   LIN {X 10.637, Y -21.360, Z 102.000}
   LaserEnd_Ext()
   LIN {X 11.146, Y -20.360, Z 102.000}
   LaserStart_Ext()
   LIN {X 9.029, Y -20.360, Z 102.000}
   LaserEnd_Ext()
   LIN {X -1.745, Y -20.360, Z 102.000}
   LaserStart_Ext()
   LIN {X -3.794, Y -20.360, Z 102.000}
   LaserEnd_Ext()
   LIN {X -4.048, Y -19.360, Z 102.000}
   LaserStart_Ext()
   LIN {X -2.060, Y -19.360, Z 102.000}
   LaserEnd_Ext()
   LIN {X 9.299, Y -19.360, Z 102.000}
   LaserStart_Ext()
   LIN {X 11.371, Y -19.360, Z 102.000}
   LaserEnd_Ext()
   LIN {X 11.596, Y -18.360, Z 102.000}
   LaserStart_Ext()
   LIN {X 9.570, Y -18.360, Z 102.000}
   LaserEnd_Ext()
   LIN {X -2.335, Y -18.360, Z 102.000}
   LaserStart_Ext()
   LIN {X -4.308, Y -18.360, Z 102.000}
   LaserEnd_Ext()
   LIN {X -4.240, Y -17.360, Z 102.000}
   LaserStart_Ext()
   LIN {X -2.147, Y -17.360, Z 102.000}
   LaserEnd_Ext()
   LIN {X 9.558, Y -17.360, Z 102.000}
   LaserStart_Ext()
   LIN {X 11.679, Y -17.360, Z 102.000}
   LaserEnd_Ext()
   LIN {X 11.721, Y -16.360, Z 102.000}
   LaserStart_Ext()
   LIN {X 9.366, Y -16.360, Z 102.000}
   LaserEnd_Ext()
   LIN {X -1.926, Y -16.360, Z 102.000}
   LaserStart_Ext()
   LIN {X -4.108, Y -16.360, Z 102.000}
   LaserEnd_Ext()
   LIN {X -3.973, Y -15.360, Z 102.000}
   LaserStart_Ext()
   LIN {X -1.705, Y -15.360, Z 102.000}
   LaserEnd_Ext()
   LIN {X 9.145, Y -15.360, Z 102.000}
   LaserStart_Ext()
   LIN {X 11.764, Y -15.360, Z 102.000}
   LaserEnd_Ext()
   LIN {X 11.791, Y -14.360, Z 102.000}
   LaserStart_Ext()
   LIN {X 8.388, Y -14.360, Z 102.000}
   LaserEnd_Ext()
   LIN {X -1.169, Y -14.360, Z 102.000}
   LaserStart_Ext()
   LIN {X -3.678, Y -14.360, Z 102.000}
   LaserEnd_Ext()
   LIN {X -3.386, Y -13.360, Z 102.000}
   LaserStart_Ext()
   LIN {X -0.277, Y -13.360, Z 102.000}
   LaserEnd_Ext()
   LIN {X 7.590, Y -13.360, Z 102.000}
   LaserStart_Ext()
   LIN {X 11.806, Y -13.360, Z 102.000}
   LaserEnd_Ext()
   LIN {X 11.817, Y -12.360, Z 102.000}
   LaserStart_Ext()
   LIN {X 5.937, Y -12.360, Z 102.000}
   LaserEnd_Ext()
   LIN {X 1.421, Y -12.360, Z 102.000}
   LaserStart_Ext()
   LIN {X -3.094, Y -12.360, Z 102.000}
   LaserEnd_Ext()
   LIN {X -2.845, Y -11.360, Z 102.000}
   LaserStart_Ext()
   LIN {X 11.809, Y -11.360, Z 102.000}
   LaserEnd_Ext()
   LIN {X 11.793, Y -10.360, Z 102.000}
   LaserStart_Ext()
   LIN {X -2.605, Y -10.360, Z 102.000}
   LaserEnd_Ext()
   LIN {X -2.364, Y -9.360, Z 102.000}
   LaserStart_Ext()
   LIN {X 11.776, Y -9.360, Z 102.000}
   LaserEnd_Ext()
   LIN {X 11.758, Y -8.360, Z 102.000}
   LaserStart_Ext()
   LIN {X -2.129, Y -8.360, Z 102.000}
   LaserEnd_Ext()
   LIN {X -1.924, Y -7.360, Z 102.000}
   LaserStart_Ext()
   LIN {X 11.706, Y -7.360, Z 102.000}
   LaserEnd_Ext()
   LIN {X 11.652, Y -6.360, Z 102.000}
   LaserStart_Ext()
   LIN {X -1.769, Y -6.360, Z 102.000}
   LaserEnd_Ext()
   LIN {X -1.619, Y -5.360, Z 102.000}
   LaserStart_Ext()
   LIN {X 11.597, Y -5.360, Z 102.000}
   LaserEnd_Ext()
   LIN {X 11.543, Y -4.360, Z 102.000}
   LaserStart_Ext()
   LIN {X -1.468, Y -4.360, Z 102.000}
   LaserEnd_Ext()
   LIN {X -1.317, Y -3.360, Z 102.000}
   LaserStart_Ext()
   LIN {X 11.470, Y -3.360, Z 102.000}
   LaserEnd_Ext()
   LIN {X 11.369, Y -2.360, Z 102.000}
   LaserStart_Ext()
   LIN {X -1.166, Y -2.360, Z 102.000}
   LaserEnd_Ext()
   LIN {X -1.015, Y -1.360, Z 102.000}
   LaserStart_Ext()
   LIN {X 11.269, Y -1.360, Z 102.000}
   LaserEnd_Ext()
   LIN {X 11.168, Y -0.360, Z 102.000}
   LaserStart_Ext()
   LIN {X -0.870, Y -0.360, Z 102.000}
   LaserEnd_Ext()
   LIN {X -0.832, Y 0.640, Z 102.000}
   LaserStart_Ext()
   LIN {X 11.068, Y 0.640, Z 102.000}
   LaserEnd_Ext()
   LIN {X 10.962, Y 1.640, Z 102.000}
   LaserStart_Ext()
   LIN {X -0.795, Y 1.640, Z 102.000}
   LaserEnd_Ext()
   LIN {X -0.758, Y 2.640, Z 102.000}
   LaserStart_Ext()
   LIN {X 10.799, Y 2.640, Z 102.000}
   LaserEnd_Ext()
   LIN {X 10.635, Y 3.640, Z 102.000}
   LaserStart_Ext()
   LIN {X -0.721, Y 3.640, Z 102.000}
   LaserEnd_Ext()
   LIN {X -0.684, Y 4.640, Z 102.000}
   LaserStart_Ext()
   LIN {X 10.471, Y 4.640, Z 102.000}
   LaserEnd_Ext()
   LIN {X 10.308, Y 5.640, Z 102.000}
   LaserStart_Ext()
   LIN {X -0.647, Y 5.640, Z 102.000}
   LaserEnd_Ext()
   LIN {X -0.610, Y 6.640, Z 102.000}
   LaserStart_Ext()
   LIN {X 10.144, Y 6.640, Z 102.000}
   LaserEnd_Ext()
   LIN {X 9.981, Y 7.640, Z 102.000}
   LaserStart_Ext()
   LIN {X -0.570, Y 7.640, Z 102.000}
   LaserEnd_Ext()
   LIN {X -0.514, Y 8.640, Z 102.000}
   LaserStart_Ext()
   LIN {X 9.817, Y 8.640, Z 102.000}
   LaserEnd_Ext()
   LIN {X 9.654, Y 9.640, Z 102.000}
   LaserStart_Ext()
   LIN {X -0.579, Y 9.640, Z 102.000}
   LaserEnd_Ext()
   LIN {X -0.671, Y 10.640, Z 102.000}
   LaserStart_Ext()
   LIN {X 9.429, Y 10.640, Z 102.000}
   LaserEnd_Ext()
   LIN {X 9.178, Y 11.640, Z 102.000}
   LaserStart_Ext()
   LIN {X -0.763, Y 11.640, Z 102.000}
   LaserEnd_Ext()
   LIN {X -0.856, Y 12.640, Z 102.000}
   LaserStart_Ext()
   LIN {X 8.927, Y 12.640, Z 102.000}
   LaserEnd_Ext()
   LIN {X 8.677, Y 13.640, Z 102.000}
   LaserStart_Ext()
   LIN {X -0.948, Y 13.640, Z 102.000}
   LaserEnd_Ext()
   LIN {X -1.040, Y 14.640, Z 102.000}
   LaserStart_Ext()
   LIN {X 8.426, Y 14.640, Z 102.000}
   LaserEnd_Ext()
   LIN {X 8.175, Y 15.640, Z 102.000}
   LaserStart_Ext()
   LIN {X -1.132, Y 15.640, Z 102.000}
   LaserEnd_Ext()
   LIN {X -1.224, Y 16.640, Z 102.000}
   LaserStart_Ext()
   LIN {X 7.925, Y 16.640, Z 102.000}
   LaserEnd_Ext()
   LIN {X 7.674, Y 17.640, Z 102.000}
   LaserStart_Ext()
   LIN {X -1.316, Y 17.640, Z 102.000}
   LaserEnd_Ext()
   LIN {X -1.415, Y 18.640, Z 102.000}
   LaserStart_Ext()
   LIN {X 7.428, Y 18.640, Z 102.000}
   LaserEnd_Ext()
   LIN {X 7.127, Y 19.640, Z 102.000}
   LaserStart_Ext()
   LIN {X -1.612, Y 19.640, Z 102.000}
   LaserEnd_Ext()
   LIN {X -1.838, Y 20.640, Z 102.000}
   LaserStart_Ext()
   LIN {X 6.799, Y 20.640, Z 102.000}
   LaserEnd_Ext()
   LIN {X 6.471, Y 21.640, Z 102.000}
   LaserStart_Ext()
   LIN {X -2.067, Y 21.640, Z 102.000}
   LaserEnd_Ext()
   LIN {X -2.296, Y 22.640, Z 102.000}
   LaserStart_Ext()
   LIN {X 6.144, Y 22.640, Z 102.000}
   LaserEnd_Ext()
   LIN {X 5.816, Y 23.640, Z 102.000}
   LaserStart_Ext()
   LIN {X -2.517, Y 23.640, Z 102.000}
   LaserEnd_Ext()
   LIN {X -2.736, Y 24.640, Z 102.000}
   LaserStart_Ext()
   LIN {X 5.488, Y 24.640, Z 102.000}
   LaserEnd_Ext()
   LIN {X 5.127, Y 25.640, Z 102.000}
   LaserStart_Ext()
   LIN {X -2.954, Y 25.640, Z 102.000}
   LaserEnd_Ext()
   LIN {X -3.172, Y 26.640, Z 102.000}
   LaserStart_Ext()
   LIN {X 4.720, Y 26.640, Z 102.000}
   LaserEnd_Ext()
   LIN {X 4.318, Y 27.640, Z 102.000}
   LaserStart_Ext()
   LIN {X -3.438, Y 27.640, Z 102.000}
   LaserEnd_Ext()
   LIN {X -3.758, Y 28.640, Z 102.000}
   LaserStart_Ext()
   LIN {X 3.920, Y 28.640, Z 102.000}
   LaserEnd_Ext()
   LIN {X 3.523, Y 29.640, Z 102.000}
   LaserStart_Ext()
   LIN {X -4.103, Y 29.640, Z 102.000}
   LaserEnd_Ext()
   LIN {X -4.447, Y 30.640, Z 102.000}
   LaserStart_Ext()
   LIN {X 3.126, Y 30.640, Z 102.000}
   LaserEnd_Ext()
   LIN {X 2.729, Y 31.640, Z 102.000}
   LaserStart_Ext()
   LIN {X -4.791, Y 31.640, Z 102.000}
   LaserEnd_Ext()
   LIN {X -5.135, Y 32.640, Z 102.000}
   LaserStart_Ext()
   LIN {X 2.275, Y 32.640, Z 102.000}
   LaserEnd_Ext()
   LIN {X 1.799, Y 33.640, Z 102.000}
   LaserStart_Ext()
   LIN {X -5.479, Y 33.640, Z 102.000}
   LaserEnd_Ext()
   LIN {X -5.852, Y 34.640, Z 102.000}
   LaserStart_Ext()
   LIN {X 1.322, Y 34.640, Z 102.000}
   LaserEnd_Ext()
   LIN {X 0.845, Y 35.640, Z 102.000}
   LaserStart_Ext()
   LIN {X -6.264, Y 35.640, Z 102.000}
   LaserEnd_Ext()
   LIN {X -6.689, Y 36.640, Z 102.000}
   LaserStart_Ext()
   LIN {X 0.377, Y 36.640, Z 102.000}
   LaserEnd_Ext()
   LIN {X -0.088, Y 37.640, Z 102.000}
   LaserStart_Ext()
   LIN {X -7.139, Y 37.640, Z 102.000}
   LaserEnd_Ext()
   LIN {X -7.596, Y 38.640, Z 102.000}
   LaserStart_Ext()
   LIN {X -0.595, Y 38.640, Z 102.000}
   LaserEnd_Ext()
   LIN {X -1.126, Y 39.640, Z 102.000}
   LaserStart_Ext()
   LIN {X -8.075, Y 39.640, Z 102.000}
   LaserEnd_Ext()
   LIN {X -8.570, Y 40.640, Z 102.000}
   LaserStart_Ext()
   LIN {X -1.658, Y 40.640, Z 102.000}
   LaserEnd_Ext()
   LIN {X -2.209, Y 41.640, Z 102.000}
   LaserStart_Ext()
   LIN {X -9.044, Y 41.640, Z 102.000}
   LaserEnd_Ext()
   LIN {X -9.321, Y 42.640, Z 102.000}
   LaserStart_Ext()
   LIN {X -2.776, Y 42.640, Z 102.000}
   LaserEnd_Ext()
   LIN {X -3.351, Y 43.640, Z 102.000}
   LaserStart_Ext()
   LIN {X -9.262, Y 43.640, Z 102.000}
   LaserEnd_Ext()
   LIN {X -8.767, Y 44.640, Z 102.000}
   LaserStart_Ext()
   LIN {X -4.018, Y 44.640, Z 102.000}
   LaserEnd_Ext()
   LIN {X -5.379, Y 45.640, Z 102.000}
   LaserStart_Ext()
   LIN {X -7.287, Y 45.640, Z 102.000}
   LaserEnd_Ext()
   LIN {X 8.308, Y -15.696, Z 102.850}
   LaserStart_Ext()
   LIN {X 8.623, Y -17.320, Z 102.850} C_DIS
   LIN {X 8.731, Y -17.865, Z 102.850} C_DIS
   LIN {X 8.484, Y -18.785, Z 102.850} C_DIS
   LIN {X 8.129, Y -20.099, Z 102.850} C_DIS
   LIN {X 7.516, Y -20.821, Z 102.850} C_DIS
   LIN {X 6.760, Y -21.715, Z 102.850} C_DIS
   LIN {X 6.064, Y -22.041, Z 102.850} C_DIS
   LIN {X 4.773, Y -22.638, Z 102.850} C_DIS
   LIN {X 2.724, Y -22.656, Z 102.850} C_DIS
   LIN {X 0.775, Y -21.816, Z 102.850} C_DIS
   LIN {X -0.300, Y -20.630, Z 102.850} C_DIS
   LIN {X -0.622, Y -20.272, Z 102.850} C_DIS
   LIN {X -0.779, Y -19.772, Z 102.850} C_DIS
   LIN {X -1.255, Y -18.283, Z 102.850} C_DIS
   LIN {X -0.812, Y -16.230, Z 102.850} C_DIS
   LIN {X -0.598, Y -15.259, Z 102.850} C_DIS
   LIN {X 0.773, Y -13.724, Z 102.850} C_DIS
   LIN {X 2.697, Y -12.858, Z 102.850} C_DIS
   LIN {X 2.949, Y -12.855, Z 102.850} C_DIS
   LIN {X 4.778, Y -12.842, Z 102.850} C_DIS
   LIN {X 6.082, Y -13.430, Z 102.850} C_DIS
   LIN {X 6.717, Y -13.713, Z 102.850} C_DIS
   LIN {X 7.260, Y -14.387, Z 102.850} C_DIS
   LIN {X 8.308, Y -15.696, Z 102.850}
   LaserEnd_Ext()
   LIN {X -1.415, Y 42.216, Z 102.850}
   LaserStart_Ext()
   LIN {X -2.278, Y 43.732, Z 102.850} C_DIS
   LIN {X -3.018, Y 44.983, Z 102.850} C_DIS
   LIN {X -4.011, Y 46.108, Z 102.850} C_DIS
   LIN {X -5.180, Y 46.661, Z 102.850} C_DIS
   LIN {X -5.583, Y 46.851, Z 102.850} C_DIS
   LIN {X -6.280, Y 46.852, Z 102.850} C_DIS
   LIN {X -7.328, Y 46.856, Z 102.850} C_DIS
   LIN {X -9.170, Y 45.752, Z 102.850} C_DIS
   LIN {X -9.479, Y 45.566, Z 102.850} C_DIS
   LIN {X -9.536, Y 45.458, Z 102.850} C_DIS
   LIN {X -10.302, Y 44.013, Z 102.850} C_DIS
   LIN {X -10.392, Y 42.442, Z 102.850} C_DIS
   LIN {X -10.380, Y 42.341, Z 102.850} C_DIS
   LIN {X -9.964, Y 41.103, Z 102.850} C_DIS
   LIN {X -9.540, Y 40.270, Z 102.850} C_DIS
   LIN {X -9.398, Y 39.988, Z 102.850} C_DIS
   LIN {X -9.127, Y 39.438, Z 102.850} C_DIS
   LIN {X -8.690, Y 38.554, Z 102.850} C_DIS
   LIN {X -8.156, Y 37.386, Z 102.850} C_DIS
   LIN {X -7.011, Y 34.771, Z 102.850} C_DIS
   LIN {X -6.857, Y 34.406, Z 102.850} C_DIS
   LIN {X -6.812, Y 34.300, Z 102.850} C_DIS
   LIN {X -6.621, Y 33.797, Z 102.850} C_DIS
   LIN {X -4.405, Y 27.356, Z 102.850} C_DIS
   LIN {X -4.262, Y 26.870, Z 102.850} C_DIS
   LIN {X -3.855, Y 25.003, Z 102.850} C_DIS
   LIN {X -2.683, Y 19.878, Z 102.850} C_DIS
   LIN {X -2.349, Y 18.189, Z 102.850} C_DIS
   LIN {X -1.587, Y 9.911, Z 102.850} C_DIS
   LIN {X -1.485, Y 8.436, Z 102.850} C_DIS
   LIN {X -1.618, Y 6.072, Z 102.850} C_DIS
   LIN {X -1.866, Y -0.630, Z 102.850} C_DIS
   LIN {X -2.699, Y -6.156, Z 102.850} C_DIS
   LIN {X -2.928, Y -7.587, Z 102.850} C_DIS
   LIN {X -3.365, Y -9.502, Z 102.850} C_DIS
   LIN {X -3.889, Y -11.680, Z 102.850} C_DIS
   LIN {X -4.676, Y -14.377, Z 102.850} C_DIS
   LIN {X -4.875, Y -15.079, Z 102.850} C_DIS
   LIN {X -4.928, Y -15.498, Z 102.850} C_DIS
   LIN {X -5.287, Y -18.223, Z 102.850} C_DIS
   LIN {X -4.582, Y -20.928, Z 102.850} C_DIS
   LIN {X -4.358, Y -21.816, Z 102.850} C_DIS
   LIN {X -3.835, Y -22.545, Z 102.850} C_DIS
   LIN {X -2.637, Y -24.194, Z 102.850} C_DIS
   LIN {X 0.472, Y -26.123, Z 102.850} C_DIS
   LIN {X 0.745, Y -26.287, Z 102.850} C_DIS
   LIN {X 1.115, Y -26.266, Z 102.850} C_DIS
   LIN {X 7.358, Y -25.978, Z 102.850} C_DIS
   LIN {X 9.637, Y -24.453, Z 102.850} C_DIS
   LIN {X 9.904, Y -24.271, Z 102.850} C_DIS
   LIN {X 10.498, Y -23.393, Z 102.850} C_DIS
   LIN {X 12.082, Y -21.065, Z 102.850} C_DIS
   LIN {X 12.379, Y -19.746, Z 102.850} C_DIS
   LIN {X 12.724, Y -18.174, Z 102.850} C_DIS
   LIN {X 12.853, Y -14.926, Z 102.850} C_DIS
   LIN {X 12.887, Y -11.955, Z 102.850} C_DIS
   LIN {X 12.850, Y -9.706, Z 102.850} C_DIS
   LIN {X 12.813, Y -8.151, Z 102.850} C_DIS
   LIN {X 12.757, Y -7.178, Z 102.850} C_DIS
   LIN {X 12.580, Y -3.931, Z 102.850} C_DIS
   LIN {X 12.129, Y 0.556, Z 102.850} C_DIS
   LIN {X 12.045, Y 1.429, Z 102.850} C_DIS
   LIN {X 11.784, Y 3.052, Z 102.850} C_DIS
   LIN {X 10.665, Y 9.895, Z 102.850} C_DIS
   LIN {X 9.253, Y 15.529, Z 102.850} C_DIS
   LIN {X 8.400, Y 18.999, Z 102.850} C_DIS
   LIN {X 8.088, Y 19.951, Z 102.850} C_DIS
   LIN {X 6.298, Y 25.412, Z 102.850} C_DIS
   LIN {X 5.919, Y 26.353, Z 102.850} C_DIS
   LIN {X 4.699, Y 29.353, Z 102.850} C_DIS
   LIN {X 3.449, Y 32.499, Z 102.850} C_DIS
   LIN {X 1.193, Y 37.232, Z 102.850} C_DIS
   LIN {X 0.717, Y 38.255, Z 102.850} C_DIS
   LIN {X 0.123, Y 39.372, Z 102.850} C_DIS
   LIN {X -1.030, Y 41.537, Z 102.850} C_DIS
   LIN {X -1.415, Y 42.216, Z 102.850}
   LaserEnd_Ext()
   LIN {X 11.602, Y -18.623, Z 102.850}
   LaserStart_Ext()
   LIN {X 11.602, Y -4.360, Z 102.850}
   LaserEnd_Ext()
   LIN {X 10.602, Y 4.086, Z 102.850}
   LaserStart_Ext()
   LIN {X 10.602, Y -21.462, Z 102.850}
   LaserEnd_Ext()
   LIN {X 9.602, Y -22.932, Z 102.850}
   LaserStart_Ext()
   LIN {X 9.602, Y -18.476, Z 102.850}
   LaserEnd_Ext()
   LIN {X 9.602, Y -17.114, Z 102.850}
   LaserStart_Ext()
   LIN {X 9.602, Y 10.024, Z 102.850}
   LaserEnd_Ext()
   LIN {X 8.602, Y 14.014, Z 102.850}
   LaserStart_Ext()
   LIN {X 8.602, Y -14.463, Z 102.850}
   LaserEnd_Ext()
   LIN {X 8.602, Y -21.087, Z 102.850}
   LaserStart_Ext()
   LIN {X 8.602, Y -23.942, Z 102.850}
   LaserEnd_Ext()
   LIN {X 7.602, Y -24.611, Z 102.850}
   LaserStart_Ext()
   LIN {X 7.602, Y -22.268, Z 102.850}
   LaserEnd_Ext()
   LIN {X 7.602, Y -13.218, Z 102.850}
   LaserStart_Ext()
   LIN {X 7.602, Y 18.058, Z 102.850}
   LaserEnd_Ext()
   LIN {X 6.602, Y 21.274, Z 102.850}
   LaserStart_Ext()
   LIN {X 6.602, Y -12.567, Z 102.850}
   LaserEnd_Ext()
   LIN {X 6.602, Y -22.893, Z 102.850}
   LaserStart_Ext()
   LIN {X 6.602, Y -25.012, Z 102.850}
   LaserEnd_Ext()
   LIN {X 5.602, Y -25.058, Z 102.850}
   LaserStart_Ext()
   LIN {X 5.602, Y -23.357, Z 102.850}
   LaserEnd_Ext()
   LIN {X 5.602, Y -12.116, Z 102.850}
   LaserStart_Ext()
   LIN {X 5.602, Y 24.326, Z 102.850}
   LaserEnd_Ext()
   LIN {X 4.602, Y 26.937, Z 102.850}
   LaserStart_Ext()
   LIN {X 4.602, Y -11.843, Z 102.850}
   LaserEnd_Ext()
   LIN {X 4.602, Y -23.640, Z 102.850}
   LaserStart_Ext()
   LIN {X 4.602, Y -25.104, Z 102.850}
   LaserEnd_Ext()
   LIN {X 3.602, Y -25.150, Z 102.850}
   LaserStart_Ext()
   LIN {X 3.602, Y -23.648, Z 102.850}
   LaserEnd_Ext()
   LIN {X 3.602, Y -11.850, Z 102.850}
   LaserStart_Ext()
   LIN {X 3.602, Y 29.406, Z 102.850}
   LaserEnd_Ext()
   LIN {X 2.602, Y 31.924, Z 102.850}
   LaserStart_Ext()
   LIN {X 2.602, Y -11.863, Z 102.850}
   LaserEnd_Ext()
   LIN {X 2.602, Y -23.653, Z 102.850}
   LaserStart_Ext()
   LIN {X 2.602, Y -25.196, Z 102.850}
   LaserEnd_Ext()
   LIN {X 1.602, Y -25.242, Z 102.850}
   LaserStart_Ext()
   LIN {X 1.602, Y -23.278, Z 102.850}
   LaserEnd_Ext()
   LIN {X 1.602, Y -12.254, Z 102.850}
   LaserStart_Ext()
   LIN {X 1.602, Y 34.050, Z 102.850}
   LaserEnd_Ext()
   LIN {X 0.602, Y 36.148, Z 102.850}
   LaserStart_Ext()
   LIN {X 0.602, Y -12.704, Z 102.850}
   LaserEnd_Ext()
   LIN {X 0.602, Y -22.834, Z 102.850}
   LaserStart_Ext()
   LIN {X 0.602, Y -25.027, Z 102.850}
   LaserEnd_Ext()
   LIN {X -0.398, Y -24.406, Z 102.850}
   LaserStart_Ext()
   LIN {X -0.398, Y -22.011, Z 102.850}
   LaserEnd_Ext()
   LIN {X -0.398, Y -13.534, Z 102.850}
   LaserStart_Ext()
   LIN {X -0.398, Y 38.223, Z 102.850}
   LaserEnd_Ext()
   LIN {X -1.398, Y 40.101, Z 102.850}
   LaserStart_Ext()
   LIN {X -1.398, Y 18.533, Z 102.850}
   LaserEnd_Ext()
   LIN {X -1.398, Y -4.232, Z 102.850}
   LaserStart_Ext()
   LIN {X -1.398, Y -14.661, Z 102.850}
   LaserEnd_Ext()
   LIN {X -1.398, Y -20.900, Z 102.850}
   LaserStart_Ext()
   LIN {X -1.398, Y -23.786, Z 102.850}
   LaserEnd_Ext()
   LIN {X -2.398, Y -22.821, Z 102.850}
   LaserStart_Ext()
   LIN {X -2.398, Y -9.757, Z 102.850}
   LaserEnd_Ext()
   LIN {X -2.398, Y 23.118, Z 102.850}
   LaserStart_Ext()
   LIN {X -2.398, Y 41.922, Z 102.850}
   LaserEnd_Ext()
   LIN {X -3.398, Y 43.661, Z 102.850}
   LaserStart_Ext()
   LIN {X -3.398, Y 27.477, Z 102.850}
   LaserEnd_Ext()
   LIN {X -3.398, Y -13.567, Z 102.850}
   LaserStart_Ext()
   LIN {X -3.398, Y -21.439, Z 102.850}
   LaserEnd_Ext()
   LIN {X -4.398, Y 30.410, Z 102.850}
   LaserStart_Ext()
   LIN {X -4.398, Y 45.038, Z 102.850}
   LaserEnd_Ext()
   LIN {X -5.398, Y 45.658, Z 102.850}
   LaserStart_Ext()
   LIN {X -5.398, Y 33.316, Z 102.850}
   LaserEnd_Ext()
   LIN {X -6.398, Y 35.864, Z 102.850}
   LaserStart_Ext()
   LIN {X -6.398, Y 45.853, Z 102.850}
   LaserEnd_Ext()
   LIN {X -7.398, Y 45.648, Z 102.850}
   LaserStart_Ext()
   LIN {X -7.398, Y 38.134, Z 102.850}
   LaserEnd_Ext()
   LIN {X -8.398, Y 40.222, Z 102.850}
   LaserStart_Ext()
   LIN {X -8.398, Y 45.048, Z 102.850}
   LaserEnd_Ext()
   LIN {X 4.939, Y -12.822, Z 103.700}
   LaserStart_Ext()
   LIN {X 6.787, Y -13.647, Z 103.700} C_DIS
   LIN {X 8.371, Y -15.609, Z 103.700} C_DIS
   LIN {X 8.811, Y -17.794, Z 103.700} C_DIS
   LIN {X 8.375, Y -19.421, Z 103.700} C_DIS
   LIN {X 8.211, Y -20.037, Z 103.700} C_DIS
   LIN {X 7.813, Y -20.509, Z 103.700} C_DIS
   LIN {X 6.849, Y -21.649, Z 103.700} C_DIS
   LIN {X 5.004, Y -22.513, Z 103.700} C_DIS
   LIN {X 4.865, Y -22.577, Z 103.700} C_DIS
   LIN {X 4.645, Y -22.579, Z 103.700} C_DIS
   LIN {X 2.756, Y -22.599, Z 103.700} C_DIS
   LIN {X 1.582, Y -22.083, Z 103.700} C_DIS
   LIN {X 0.865, Y -21.764, Z 103.700} C_DIS
   LIN {X 0.170, Y -20.996, Z 103.700} C_DIS
   LIN {X -0.536, Y -20.222, Z 103.700} C_DIS
   LIN {X -0.829, Y -19.314, Z 103.700} C_DIS
   LIN {X -1.173, Y -18.236, Z 103.700} C_DIS
   LIN {X -0.778, Y -16.404, Z 103.700} C_DIS
   LIN {X -0.524, Y -15.212, Z 103.700} C_DIS
   LIN {X 0.151, Y -14.458, Z 103.700} C_DIS
   LIN {X 0.871, Y -13.652, Z 103.700} C_DIS
   LIN {X 2.757, Y -12.803, Z 103.700} C_DIS
   LIN {X 4.718, Y -12.781, Z 103.700} C_DIS
   LIN {X 4.847, Y -12.780, Z 103.700} C_DIS
   LIN {X 4.939, Y -12.822, Z 103.700}
   LaserEnd_Ext()
   LIN {X 12.805, Y -18.094, Z 103.700}
   LaserStart_Ext()
   LIN {X 12.887, Y -16.043, Z 103.700} C_DIS
   LIN {X 12.927, Y -14.834, Z 103.700} C_DIS
   LIN {X 12.939, Y -13.141, Z 103.700} C_DIS
   LIN {X 12.953, Y -11.875, Z 103.700} C_DIS
   LIN {X 12.937, Y -10.915, Z 103.700} C_DIS
   LIN {X 12.871, Y -8.071, Z 103.700} C_DIS
   LIN {X 12.767, Y -6.290, Z 103.700} C_DIS
   LIN {X 12.652, Y -4.177, Z 103.700} C_DIS
   LIN {X 12.359, Y -1.255, Z 103.700} C_DIS
   LIN {X 12.136, Y 1.075, Z 103.700} C_DIS
   LIN {X 11.440, Y 5.404, Z 103.700} C_DIS
   LIN {X 10.744, Y 9.656, Z 103.700} C_DIS
   LIN {X 9.867, Y 13.155, Z 103.700} C_DIS
   LIN {X 8.490, Y 18.760, Z 103.700} C_DIS
   LIN {X 7.986, Y 20.296, Z 103.700} C_DIS
   LIN {X 6.350, Y 25.289, Z 103.700} C_DIS
   LIN {X 5.786, Y 26.686, Z 103.700} C_DIS
   LIN {X 3.974, Y 31.142, Z 103.700} C_DIS
   LIN {X 3.369, Y 32.666, Z 103.700} C_DIS
   LIN {X 0.987, Y 37.662, Z 103.700} C_DIS
   LIN {X 0.802, Y 38.048, Z 103.700} C_DIS
   LIN {X 0.689, Y 38.260, Z 103.700} C_DIS
   LIN {X -1.033, Y 41.492, Z 103.700} C_DIS
   LIN {X -2.132, Y 43.416, Z 103.700} C_DIS
   LIN {X -2.338, Y 43.779, Z 103.700} C_DIS
   LIN {X -2.415, Y 43.909, Z 103.700} C_DIS
   LIN {X -3.097, Y 45.052, Z 103.700} C_DIS
   LIN {X -3.968, Y 46.028, Z 103.700} C_DIS
   LIN {X -4.076, Y 46.150, Z 103.700} C_DIS
   LIN {X -4.304, Y 46.256, Z 103.700} C_DIS
   LIN {X -5.651, Y 46.889, Z 103.700} C_DIS
   LIN {X -7.396, Y 46.889, Z 103.700} C_DIS
   LIN {X -8.094, Y 46.467, Z 103.700} C_DIS
   LIN {X -9.539, Y 45.599, Z 103.700} C_DIS
   LIN {X -10.345, Y 44.074, Z 103.700} C_DIS
   LIN {X -10.453, Y 42.422, Z 103.700} C_DIS
   LIN {X -10.037, Y 41.186, Z 103.700} C_DIS
   LIN {X -9.983, Y 41.062, Z 103.700} C_DIS
   LIN {X -9.449, Y 40.018, Z 103.700} C_DIS
   LIN {X -9.064, Y 39.246, Z 103.700} C_DIS
   LIN {X -8.737, Y 38.585, Z 103.700} C_DIS
   LIN {X -8.538, Y 38.149, Z 103.700} C_DIS
   LIN {X -7.601, Y 36.008, Z 103.700} C_DIS
   LIN {X -6.796, Y 34.195, Z 103.700} C_DIS
   LIN {X -6.677, Y 33.903, Z 103.700} C_DIS
   LIN {X -4.322, Y 27.037, Z 103.700} C_DIS
   LIN {X -4.289, Y 26.933, Z 103.700} C_DIS
   LIN {X -2.760, Y 20.246, Z 103.700} C_DIS
   LIN {X -2.305, Y 17.940, Z 103.700} C_DIS
   LIN {X -1.611, Y 10.405, Z 103.700} C_DIS
   LIN {X -1.458, Y 8.186, Z 103.700} C_DIS
   LIN {X -1.657, Y 4.629, Z 103.700} C_DIS
   LIN {X -1.864, Y -0.951, Z 103.700} C_DIS
   LIN {X -2.558, Y -5.552, Z 103.700} C_DIS
   LIN {X -2.894, Y -7.654, Z 103.700} C_DIS
   LIN {X -3.536, Y -10.467, Z 103.700} C_DIS
   LIN {X -3.765, Y -11.420, Z 103.700} C_DIS
   LIN {X -4.110, Y -12.600, Z 103.700} C_DIS
   LIN {X -4.802, Y -15.040, Z 103.700} C_DIS
   LIN {X -4.984, Y -16.493, Z 103.700} C_DIS
   LIN {X -5.206, Y -18.184, Z 103.700} C_DIS
   LIN {X -4.383, Y -21.347, Z 103.700} C_DIS
   LIN {X -4.269, Y -21.775, Z 103.700} C_DIS
   LIN {X -4.049, Y -22.076, Z 103.700} C_DIS
   LIN {X -2.543, Y -24.150, Z 103.700} C_DIS
   LIN {X -0.667, Y -25.314, Z 103.700} C_DIS
   LIN {X 0.878, Y -26.246, Z 103.700} C_DIS
   LIN {X 2.981, Y -26.124, Z 103.700} C_DIS
   LIN {X 7.438, Y -25.919, Z 103.700} C_DIS
   LIN {X 9.066, Y -24.829, Z 103.700} C_DIS
   LIN {X 10.001, Y -24.196, Z 103.700} C_DIS
   LIN {X 12.078, Y -21.122, Z 103.700} C_DIS
   LIN {X 12.170, Y -20.986, Z 103.700} C_DIS
   LIN {X 12.805, Y -18.094, Z 103.700}
   LaserEnd_Ext()
   LIN {X -7.726, Y 45.522, Z 103.700}
   LaserStart_Ext()
   LIN {X -5.093, Y 45.522, Z 103.700}
   LaserEnd_Ext()
   LIN {X -3.963, Y 44.522, Z 103.700}
   LaserStart_Ext()
   LIN {X -8.977, Y 44.522, Z 103.700}
   LaserEnd_Ext()
   LIN {X -9.389, Y 43.522, Z 103.700}
   LaserStart_Ext()
   LIN {X -3.349, Y 43.522, Z 103.700}
   LaserEnd_Ext()
   LIN {X -2.772, Y 42.522, Z 103.700}
   LaserStart_Ext()
   LIN {X -9.432, Y 42.522, Z 103.700}
   LaserEnd_Ext()
   LIN {X -9.095, Y 41.522, Z 103.700}
   LaserStart_Ext()
   LIN {X -2.201, Y 41.522, Z 103.700}
   LaserEnd_Ext()
   LIN {X -1.649, Y 40.522, Z 103.700}
   LaserStart_Ext()
   LIN {X -8.583, Y 40.522, Z 103.700}
   LaserEnd_Ext()
   LIN {X -8.085, Y 39.522, Z 103.700}
   LaserStart_Ext()
   LIN {X -1.116, Y 39.522, Z 103.700}
   LaserEnd_Ext()
   LIN {X -0.583, Y 38.522, Z 103.700}
   LaserStart_Ext()
   LIN {X -7.610, Y 38.522, Z 103.700}
   LaserEnd_Ext()
   LIN {X -7.172, Y 37.522, Z 103.700}
   LaserStart_Ext()
   LIN {X -0.055, Y 37.522, Z 103.700}
   LaserEnd_Ext()
   LIN {X 0.423, Y 36.522, Z 103.700}
   LaserStart_Ext()
   LIN {X -6.734, Y 36.522, Z 103.700}
   LaserEnd_Ext()
   LIN {X -6.291, Y 35.522, Z 103.700}
   LaserStart_Ext()
   LIN {X 0.899, Y 35.522, Z 103.700}
   LaserEnd_Ext()
   LIN {X 1.376, Y 34.522, Z 103.700}
   LaserStart_Ext()
   LIN {X -5.849, Y 34.522, Z 103.700}
   LaserEnd_Ext()
   LIN {X -5.489, Y 33.522, Z 103.700}
   LaserStart_Ext()
   LIN {X 1.853, Y 33.522, Z 103.700}
   LaserEnd_Ext()
   LIN {X 2.330, Y 32.522, Z 103.700}
   LaserStart_Ext()
   LIN {X -5.146, Y 32.522, Z 103.700}
   LaserEnd_Ext()
   LIN {X -4.803, Y 31.522, Z 103.700}
   LaserStart_Ext()
   LIN {X 2.747, Y 31.522, Z 103.700}
   LaserEnd_Ext()
   LIN {X 3.147, Y 30.522, Z 103.700}
   LaserStart_Ext()
   LIN {X -4.460, Y 30.522, Z 103.700}
   LaserEnd_Ext()
   LIN {X -4.117, Y 29.522, Z 103.700}
   LaserStart_Ext()
   LIN {X 3.553, Y 29.522, Z 103.700}
   LaserEnd_Ext()
   LIN {X 3.960, Y 28.522, Z 103.700}
   LaserStart_Ext()
   LIN {X -3.774, Y 28.522, Z 103.700}
   LaserEnd_Ext()
   LIN {X -3.431, Y 27.522, Z 103.700}
   LaserStart_Ext()
   LIN {X 4.367, Y 27.522, Z 103.700}
   LaserEnd_Ext()
   LIN {X 4.774, Y 26.522, Z 103.700}
   LaserStart_Ext()
   LIN {X -3.170, Y 26.522, Z 103.700}
   LaserEnd_Ext()
   LIN {X -2.941, Y 25.522, Z 103.700}
   LaserStart_Ext()
   LIN {X 5.177, Y 25.522, Z 103.700}
   LaserEnd_Ext()
   LIN {X 5.549, Y 24.522, Z 103.700}
   LaserStart_Ext()
   LIN {X -2.712, Y 24.522, Z 103.700}
   LaserEnd_Ext()
   LIN {X -2.483, Y 23.522, Z 103.700}
   LaserStart_Ext()
   LIN {X 5.876, Y 23.522, Z 103.700}
   LaserEnd_Ext()
   LIN {X 6.204, Y 22.522, Z 103.700}
   LaserStart_Ext()
   LIN {X -2.255, Y 22.522, Z 103.700}
   LaserEnd_Ext()
   LIN {X -2.026, Y 21.522, Z 103.700}
   LaserStart_Ext()
   LIN {X 6.532, Y 21.522, Z 103.700}
   LaserEnd_Ext()
   LIN {X 6.859, Y 20.522, Z 103.700}
   LaserStart_Ext()
   LIN {X -1.797, Y 20.522, Z 103.700}
   LaserEnd_Ext()
   LIN {X -1.598, Y 19.522, Z 103.700}
   LaserStart_Ext()
   LIN {X 7.187, Y 19.522, Z 103.700}
   LaserEnd_Ext()
   LIN {X 7.516, Y 18.522, Z 103.700}
   LaserStart_Ext()
   LIN {X -1.400, Y 18.522, Z 103.700}
   LaserEnd_Ext()
   LIN {X -1.262, Y 17.522, Z 103.700}
   LaserStart_Ext()
   LIN {X 7.764, Y 17.522, Z 103.700}
   LaserEnd_Ext()
   LIN {X 8.010, Y 16.522, Z 103.700}
   LaserStart_Ext()
   LIN {X -1.170, Y 16.522, Z 103.700}
   LaserEnd_Ext()
   LIN {X -1.078, Y 15.522, Z 103.700}
   LaserStart_Ext()
   LIN {X 8.256, Y 15.522, Z 103.700}
   LaserEnd_Ext()
   LIN {X 8.502, Y 14.522, Z 103.700}
   LaserStart_Ext()
   LIN {X -0.986, Y 14.522, Z 103.700}
   LaserEnd_Ext()
   LIN {X -0.893, Y 13.522, Z 103.700}
   LaserStart_Ext()
   LIN {X 8.747, Y 13.522, Z 103.700}
   LaserEnd_Ext()
   LIN {X 8.995, Y 12.522, Z 103.700}
   LaserStart_Ext()
   LIN {X -0.801, Y 12.522, Z 103.700}
   LaserEnd_Ext()
   LIN {X -0.709, Y 11.522, Z 103.700}
   LaserStart_Ext()
   LIN {X 9.246, Y 11.522, Z 103.700}
   LaserEnd_Ext()
   LIN {X 9.496, Y 10.522, Z 103.700}
   LaserStart_Ext()
   LIN {X -0.617, Y 10.522, Z 103.700}
   LaserEnd_Ext()
   LIN {X -0.547, Y 9.522, Z 103.700}
   LaserStart_Ext()
   LIN {X 9.747, Y 9.522, Z 103.700}
   LaserEnd_Ext()
   LIN {X 9.917, Y 8.522, Z 103.700}
   LaserStart_Ext()
   LIN {X -0.479, Y 8.522, Z 103.700}
   LaserEnd_Ext()
   LIN {X -0.493, Y 7.522, Z 103.700}
   LaserStart_Ext()
   LIN {X 10.080, Y 7.522, Z 103.700}
   LaserEnd_Ext()
   LIN {X 10.244, Y 6.522, Z 103.700}
   LaserStart_Ext()
   LIN {X -0.550, Y 6.522, Z 103.700}
   LaserEnd_Ext()
   LIN {X -0.606, Y 5.522, Z 103.700}
   LaserStart_Ext()
   LIN {X 10.407, Y 5.522, Z 103.700}
   LaserEnd_Ext()
   LIN {X 10.569, Y 4.522, Z 103.700}
   LaserStart_Ext()
   LIN {X -0.661, Y 4.522, Z 103.700}
   LaserEnd_Ext()
   LIN {X -0.698, Y 3.522, Z 103.700}
   LaserStart_Ext()
   LIN {X 10.730, Y 3.522, Z 103.700}
   LaserEnd_Ext()
   LIN {X 10.890, Y 2.522, Z 103.700}
   LaserStart_Ext()
   LIN {X -0.735, Y 2.522, Z 103.700}
   LaserEnd_Ext()
   LIN {X -0.772, Y 1.522, Z 103.700}
   LaserStart_Ext()
   LIN {X 11.051, Y 1.522, Z 103.700}
   LaserEnd_Ext()
   LIN {X 11.184, Y 0.522, Z 103.700}
   LaserStart_Ext()
   LIN {X -0.809, Y 0.522, Z 103.700}
   LaserEnd_Ext()
   LIN {X -0.846, Y -0.478, Z 103.700}
   LaserStart_Ext()
   LIN {X 11.280, Y -0.478, Z 103.700}
   LaserEnd_Ext()
   LIN {X 11.376, Y -1.478, Z 103.700}
   LaserStart_Ext()
   LIN {X -0.932, Y -1.478, Z 103.700}
   LaserEnd_Ext()
   LIN {X -1.083, Y -2.478, Z 103.700}
   LaserStart_Ext()
   LIN {X 11.477, Y -2.478, Z 103.700}
   LaserEnd_Ext()
   LIN {X 11.577, Y -3.478, Z 103.700}
   LaserStart_Ext()
   LIN {X -1.234, Y -3.478, Z 103.700}
   LaserEnd_Ext()
   LIN {X -1.385, Y -4.478, Z 103.700}
   LaserStart_Ext()
   LIN {X 11.667, Y -4.478, Z 103.700}
   LaserEnd_Ext()
   LIN {X 11.722, Y -5.478, Z 103.700}
   LaserStart_Ext()
   LIN {X -1.536, Y -5.478, Z 103.700}
   LaserEnd_Ext()
   LIN {X -1.693, Y -6.478, Z 103.700}
   LaserStart_Ext()
   LIN {X 11.777, Y -6.478, Z 103.700}
   LaserEnd_Ext()
   LIN {X 11.835, Y -7.478, Z 103.700}
   LaserStart_Ext()
   LIN {X -1.853, Y -7.478, Z 103.700}
   LaserEnd_Ext()
   LIN {X -2.057, Y -8.478, Z 103.700}
   LaserStart_Ext()
   LIN {X 11.880, Y -8.478, Z 103.700}
   LaserEnd_Ext()
   LIN {X 11.903, Y -9.478, Z 103.700}
   LaserStart_Ext()
   LIN {X -2.285, Y -9.478, Z 103.700}
   LaserEnd_Ext()
   LIN {X -2.513, Y -10.478, Z 103.700}
   LaserStart_Ext()
   LIN {X 11.927, Y -10.478, Z 103.700}
   LaserEnd_Ext()
   LIN {X 11.947, Y -11.478, Z 103.700}
   LaserStart_Ext()
   LIN {X -2.751, Y -11.478, Z 103.700}
   LaserEnd_Ext()
   LIN {X -3.032, Y -12.478, Z 103.700}
   LaserStart_Ext()
   LIN {X 1.041, Y -12.478, Z 103.700}
   LaserEnd_Ext()
   LIN {X 6.623, Y -12.478, Z 103.700}
   LaserStart_Ext()
   LIN {X 11.946, Y -12.478, Z 103.700}
   LaserEnd_Ext()
   LIN {X 11.937, Y -13.478, Z 103.700}
   LaserStart_Ext()
   LIN {X 7.936, Y -13.478, Z 103.700}
   LaserEnd_Ext()
   LIN {X -0.315, Y -13.478, Z 103.700}
   LaserStart_Ext()
   LIN {X -3.319, Y -13.478, Z 103.700}
   LaserEnd_Ext()
   LIN {X -3.603, Y -14.478, Z 103.700}
   LaserStart_Ext()
   LIN {X -1.210, Y -14.478, Z 103.700}
   LaserEnd_Ext()
   LIN {X 8.743, Y -14.478, Z 103.700}
   LaserStart_Ext()
   LIN {X 11.929, Y -14.478, Z 103.700}
   LaserEnd_Ext()
   LIN {X 11.905, Y -15.478, Z 103.700}
   LaserStart_Ext()
   LIN {X 9.374, Y -15.478, Z 103.700}
   LaserEnd_Ext()
   LIN {X -1.603, Y -15.478, Z 103.700}
   LaserStart_Ext()
   LIN {X -3.849, Y -15.478, Z 103.700}
   LaserEnd_Ext()
   LIN {X -3.974, Y -16.478, Z 103.700}
   LaserStart_Ext()
   LIN {X -1.817, Y -16.478, Z 103.700}
   LaserEnd_Ext()
   LIN {X 9.571, Y -16.478, Z 103.700}
   LaserStart_Ext()
   LIN {X 11.869, Y -16.478, Z 103.700}
   LaserEnd_Ext()
   LIN {X 11.829, Y -17.478, Z 103.700}
   LaserStart_Ext()
   LIN {X 9.768, Y -17.478, Z 103.700}
   LaserEnd_Ext()
   LIN {X -2.033, Y -17.478, Z 103.700}
   LaserStart_Ext()
   LIN {X -4.105, Y -17.478, Z 103.700}
   LaserEnd_Ext()
   LIN {X -4.096, Y -18.478, Z 103.700}
   LaserStart_Ext()
   LIN {X -2.142, Y -18.478, Z 103.700}
   LaserEnd_Ext()
   LIN {X 9.663, Y -18.478, Z 103.700}
   LaserStart_Ext()
   LIN {X 11.697, Y -18.478, Z 103.700}
   LaserEnd_Ext()
   LIN {X 11.478, Y -19.478, Z 103.700}
   LaserStart_Ext()
   LIN {X 9.395, Y -19.478, Z 103.700}
   LaserEnd_Ext()
   LIN {X -1.826, Y -19.478, Z 103.700}
   LaserStart_Ext()
   LIN {X -3.836, Y -19.478, Z 103.700}
   LaserEnd_Ext()
   LIN {X -3.576, Y -20.478, Z 103.700}
   LaserStart_Ext()
   LIN {X -1.504, Y -20.478, Z 103.700}
   LaserEnd_Ext()
   LIN {X 9.107, Y -20.478, Z 103.700}
   LaserStart_Ext()
   LIN {X 11.258, Y -20.478, Z 103.700}
   LaserEnd_Ext()
   LIN {X 10.630, Y -21.478, Z 103.700}
   LaserStart_Ext()
   LIN {X 8.303, Y -21.478, Z 103.700}
   LaserEnd_Ext()
   LIN {X -0.744, Y -21.478, Z 103.700}
   LaserStart_Ext()
   LIN {X -3.247, Y -21.478, Z 103.700}
   LaserEnd_Ext()
   LIN {X -2.521, Y -22.478, Z 103.700}
   LaserStart_Ext()
   LIN {X 0.167, Y -22.478, Z 103.700}
   LaserEnd_Ext()
   LIN {X 7.405, Y -22.478, Z 103.700}
   LaserStart_Ext()
   LIN {X 9.954, Y -22.478, Z 103.700}
   LaserEnd_Ext()
   LIN {X 9.277, Y -23.478, Z 103.700}
   LaserStart_Ext()
   LIN {X 5.298, Y -23.478, Z 103.700}
   LaserEnd_Ext()
   LIN {X 2.270, Y -23.478, Z 103.700}
   LaserStart_Ext()
   LIN {X -1.728, Y -23.478, Z 103.700}
   LaserEnd_Ext()
   LIN {X -0.115, Y -24.478, Z 103.700}
   LaserStart_Ext()
   LIN {X 7.792, Y -24.478, Z 103.700}
   LaserEnd_Ext()
   LIN {X 1.667, Y -13.265, Z 104.550}
   LaserStart_Ext()
   LIN {X 2.817, Y -12.748, Z 104.550} C_DIS
   LIN {X 3.757, Y -12.737, Z 104.550} C_DIS
   LIN {X 4.915, Y -12.719, Z 104.550} C_DIS
   LIN {X 6.233, Y -13.302, Z 104.550} C_DIS
   LIN {X 6.858, Y -13.581, Z 104.550} C_DIS
   LIN {X 7.350, Y -14.191, Z 104.550} C_DIS
   LIN {X 8.459, Y -15.556, Z 104.550} C_DIS
   LIN {X 8.777, Y -17.141, Z 104.550} C_DIS
   LIN {X 8.892, Y -17.723, Z 104.550} C_DIS
   LIN {X 8.776, Y -18.156, Z 104.550} C_DIS
   LIN {X 8.292, Y -19.975, Z 104.550} C_DIS
   LIN {X 7.119, Y -21.370, Z 104.550} C_DIS
   LIN {X 6.939, Y -21.583, Z 104.550} C_DIS
   LIN {X 6.528, Y -21.775, Z 104.550} C_DIS
   LIN {X 4.948, Y -22.517, Z 104.550} C_DIS
   LIN {X 3.853, Y -22.532, Z 104.550} C_DIS
   LIN {X 2.848, Y -22.543, Z 104.550} C_DIS
   LIN {X 1.552, Y -21.973, Z 104.550} C_DIS
   LIN {X 0.955, Y -21.712, Z 104.550} C_DIS
   LIN {X 0.624, Y -21.351, Z 104.550} C_DIS
   LIN {X -0.450, Y -20.173, Z 104.550} C_DIS
   LIN {X -0.982, Y -18.523, Z 104.550} C_DIS
   LIN {X -1.092, Y -18.188, Z 104.550} C_DIS
   LIN {X -0.985, Y -17.683, Z 104.550} C_DIS
   LIN {X -0.447, Y -15.157, Z 104.550} C_DIS
   LIN {X 0.569, Y -14.022, Z 104.550} C_DIS
   LIN {X 0.948, Y -13.594, Z 104.550} C_DIS
   LIN {X 1.667, Y -13.265, Z 104.550}
   LaserEnd_Ext()
   LIN {X 10.097, Y -24.120, Z 104.550}
   LaserStart_Ext()
   LIN {X 11.470, Y -22.089, Z 104.550} C_DIS
   LIN {X 12.257, Y -20.908, Z 104.550} C_DIS
   LIN {X 12.617, Y -19.241, Z 104.550} C_DIS
   LIN {X 12.886, Y -18.014, Z 104.550} C_DIS
   LIN {X 12.920, Y -17.177, Z 104.550} C_DIS
   LIN {X 13.000, Y -14.754, Z 104.550} C_DIS
   LIN {X 13.019, Y -12.116, Z 104.550} C_DIS
   LIN {X 13.020, Y -11.794, Z 104.550} C_DIS
   LIN {X 12.995, Y -10.827, Z 104.550} C_DIS
   LIN {X 12.928, Y -7.991, Z 104.550} C_DIS
   LIN {X 12.778, Y -5.403, Z 104.550} C_DIS
   LIN {X 12.725, Y -4.422, Z 104.550} C_DIS
   LIN {X 12.588, Y -3.065, Z 104.550} C_DIS
   LIN {X 12.227, Y 0.721, Z 104.550} C_DIS
   LIN {X 11.095, Y 7.757, Z 104.550} C_DIS
   LIN {X 10.824, Y 9.416, Z 104.550} C_DIS
   LIN {X 10.481, Y 10.782, Z 104.550} C_DIS
   LIN {X 8.579, Y 18.520, Z 104.550} C_DIS
   LIN {X 7.884, Y 20.641, Z 104.550} C_DIS
   LIN {X 6.401, Y 25.166, Z 104.550} C_DIS
   LIN {X 5.653, Y 27.019, Z 104.550} C_DIS
   LIN {X 3.300, Y 32.805, Z 104.550} C_DIS
   LIN {X 0.960, Y 37.696, Z 104.550} C_DIS
   LIN {X 0.532, Y 38.518, Z 104.550} C_DIS
   LIN {X -0.556, Y 40.547, Z 104.550} C_DIS
   LIN {X -1.036, Y 41.448, Z 104.550} C_DIS
   LIN {X -1.435, Y 42.147, Z 104.550} C_DIS
   LIN {X -2.399, Y 43.824, Z 104.550} C_DIS
   LIN {X -3.138, Y 45.060, Z 104.550} C_DIS
   LIN {X -4.143, Y 46.191, Z 104.550} C_DIS
   LIN {X -5.336, Y 46.749, Z 104.550} C_DIS
   LIN {X -5.718, Y 46.927, Z 104.550} C_DIS
   LIN {X -6.373, Y 46.925, Z 104.550} C_DIS
   LIN {X -7.463, Y 46.923, Z 104.550} C_DIS
   LIN {X -9.446, Y 45.724, Z 104.550} C_DIS
   LIN {X -9.599, Y 45.632, Z 104.550} C_DIS
   LIN {X -9.689, Y 45.463, Z 104.550} C_DIS
   LIN {X -10.421, Y 44.071, Z 104.550} C_DIS
   LIN {X -10.489, Y 42.837, Z 104.550} C_DIS
   LIN {X -10.511, Y 42.458, Z 104.550} C_DIS
   LIN {X -10.407, Y 42.150, Z 104.550} C_DIS
   LIN {X -10.073, Y 41.159, Z 104.550} C_DIS
   LIN {X -9.664, Y 40.368, Z 104.550} C_DIS
   LIN {X -9.500, Y 40.047, Z 104.550} C_DIS
   LIN {X -9.151, Y 39.346, Z 104.550} C_DIS
   LIN {X -8.786, Y 38.616, Z 104.550} C_DIS
   LIN {X -8.665, Y 38.358, Z 104.550} C_DIS
   LIN {X -6.934, Y 34.461, Z 104.550} C_DIS
   LIN {X -6.549, Y 33.512, Z 104.550} C_DIS
   LIN {X -4.507, Y 27.561, Z 104.550} C_DIS
   LIN {X -4.206, Y 26.599, Z 104.550} C_DIS
   LIN {X -2.837, Y 20.614, Z 104.550} C_DIS
   LIN {X -2.260, Y 17.690, Z 104.550} C_DIS
   LIN {X -1.634, Y 10.899, Z 104.550} C_DIS
   LIN {X -1.430, Y 7.935, Z 104.550} C_DIS
   LIN {X -1.697, Y 3.185, Z 104.550} C_DIS
   LIN {X -1.862, Y -1.272, Z 104.550} C_DIS
   LIN {X -2.416, Y -4.947, Z 104.550} C_DIS
   LIN {X -2.860, Y -7.721, Z 104.550} C_DIS
   LIN {X -3.605, Y -10.984, Z 104.550} C_DIS
   LIN {X -3.665, Y -11.252, Z 104.550} C_DIS
   LIN {X -3.737, Y -11.506, Z 104.550} C_DIS
   LIN {X -4.728, Y -15.000, Z 104.550} C_DIS
   LIN {X -5.039, Y -17.489, Z 104.550} C_DIS
   LIN {X -5.126, Y -18.146, Z 104.550} C_DIS
   LIN {X -4.806, Y -19.374, Z 104.550} C_DIS
   LIN {X -4.181, Y -21.734, Z 104.550} C_DIS
   LIN {X -2.965, Y -23.394, Z 104.550} C_DIS
   LIN {X -2.449, Y -24.105, Z 104.550} C_DIS
   LIN {X -1.805, Y -24.504, Z 104.550} C_DIS
   LIN {X 1.012, Y -26.205, Z 104.550} C_DIS
   LIN {X 4.847, Y -25.982, Z 104.550} C_DIS
   LIN {X 7.519, Y -25.859, Z 104.550} C_DIS
   LIN {X 8.494, Y -25.206, Z 104.550} C_DIS
   LIN {X 10.097, Y -24.120, Z 104.550}
   LaserEnd_Ext()
   LIN {X -9.280, Y 41.937, Z 104.550}
   LaserStart_Ext()
   LIN {X -9.280, Y 44.093, Z 104.550}
   LaserEnd_Ext()
   LIN {X -8.280, Y 45.261, Z 104.550}
   LaserStart_Ext()
   LIN {X -8.280, Y 39.841, Z 104.550}
   LaserEnd_Ext()
   LIN {X -7.280, Y 37.703, Z 104.550}
   LaserStart_Ext()
   LIN {X -7.280, Y 45.865, Z 104.550}
   LaserEnd_Ext()
   LIN {X -6.280, Y 45.925, Z 104.550}
   LaserStart_Ext()
   LIN {X -6.280, Y 35.452, Z 104.550}
   LaserEnd_Ext()
   LIN {X -5.280, Y 32.894, Z 104.550}
   LaserStart_Ext()
   LIN {X -5.280, Y 45.619, Z 104.550}
   LaserEnd_Ext()
   LIN {X -4.280, Y 44.847, Z 104.550}
   LaserStart_Ext()
   LIN {X -4.280, Y 29.979, Z 104.550}
   LaserEnd_Ext()
   LIN {X -3.280, Y -21.230, Z 104.550}
   LaserStart_Ext()
   LIN {X -3.280, Y -13.560, Z 104.550}
   LaserEnd_Ext()
   LIN {X -3.280, Y 26.987, Z 104.550}
   LaserStart_Ext()
   LIN {X -3.280, Y 43.349, Z 104.550}
   LaserEnd_Ext()
   LIN {X -2.280, Y 41.609, Z 104.550}
   LaserStart_Ext()
   LIN {X -2.280, Y 22.662, Z 104.550}
   LaserEnd_Ext()
   LIN {X -2.280, Y -9.674, Z 104.550}
   LaserStart_Ext()
   LIN {X -2.280, Y -22.637, Z 104.550}
   LaserEnd_Ext()
   LIN {X -1.280, Y -23.653, Z 104.550}
   LaserStart_Ext()
   LIN {X -1.280, Y -20.729, Z 104.550}
   LaserEnd_Ext()
   LIN {X -1.280, Y -14.606, Z 104.550}
   LaserStart_Ext()
   LIN {X -1.280, Y -4.117, Z 104.550}
   LaserEnd_Ext()
   LIN {X -1.280, Y 17.888, Z 104.550}
   LaserStart_Ext()
   LIN {X -1.280, Y 39.781, Z 104.550}
   LaserEnd_Ext()
   LIN {X -0.280, Y 37.912, Z 104.550}
   LaserStart_Ext()
   LIN {X -0.280, Y -13.472, Z 104.550}
   LaserEnd_Ext()
   LIN {X -0.280, Y -21.844, Z 104.550}
   LaserStart_Ext()
   LIN {X -0.280, Y -24.257, Z 104.550}
   LaserEnd_Ext()
   LIN {X 0.720, Y -24.861, Z 104.550}
   LaserStart_Ext()
   LIN {X 0.720, Y -22.700, Z 104.550}
   LaserEnd_Ext()
   LIN {X 0.720, Y -12.599, Z 104.550}
   LaserStart_Ext()
   LIN {X 0.720, Y 35.882, Z 104.550}
   LaserEnd_Ext()
   LIN {X 1.720, Y 33.792, Z 104.550}
   LaserStart_Ext()
   LIN {X 1.720, Y -12.145, Z 104.550}
   LaserEnd_Ext()
   LIN {X 1.720, Y -23.139, Z 104.550}
   LaserStart_Ext()
   LIN {X 1.720, Y -25.162, Z 104.550}
   LaserEnd_Ext()
   LIN {X 2.720, Y -25.104, Z 104.550}
   LaserStart_Ext()
   LIN {X 2.720, Y -23.533, Z 104.550}
   LaserEnd_Ext()
   LIN {X 2.720, Y -11.753, Z 104.550}
   LaserStart_Ext()
   LIN {X 2.720, Y 31.577, Z 104.550}
   LaserEnd_Ext()
   LIN {X 3.720, Y 29.118, Z 104.550}
   LaserStart_Ext()
   LIN {X 3.720, Y -11.738, Z 104.550}
   LaserEnd_Ext()
   LIN {X 3.720, Y -23.533, Z 104.550}
   LaserStart_Ext()
   LIN {X 3.720, Y -25.046, Z 104.550}
   LaserEnd_Ext()
   LIN {X 4.720, Y -24.988, Z 104.550}
   LaserStart_Ext()
   LIN {X 4.720, Y -23.520, Z 104.550}
   LaserEnd_Ext()
   LIN {X 4.720, Y -11.722, Z 104.550}
   LaserStart_Ext()
   LIN {X 4.720, Y 26.660, Z 104.550}
   LaserEnd_Ext()
   LIN {X 5.720, Y 24.031, Z 104.550}
   LaserStart_Ext()
   LIN {X 5.720, Y -11.981, Z 104.550}
   LaserEnd_Ext()
   LIN {X 5.720, Y -23.259, Z 104.550}
   LaserStart_Ext()
   LIN {X 5.720, Y -24.941, Z 104.550}
   LaserEnd_Ext()
   LIN {X 6.720, Y -24.895, Z 104.550}
   LaserStart_Ext()
   LIN {X 6.720, Y -22.789, Z 104.550}
   LaserEnd_Ext()
   LIN {X 6.720, Y -12.424, Z 104.550}
   LaserStart_Ext()
   LIN {X 6.720, Y 20.980, Z 104.550}
   LaserEnd_Ext()
   LIN {X 7.720, Y 17.827, Z 104.550}
   LaserStart_Ext()
   LIN {X 7.720, Y -13.056, Z 104.550}
   LaserEnd_Ext()
   LIN {X 7.720, Y -22.207, Z 104.550}
   LaserStart_Ext()
   LIN {X 7.720, Y -24.521, Z 104.550}
   LaserEnd_Ext()
   LIN {X 8.720, Y -23.845, Z 104.550}
   LaserStart_Ext()
   LIN {X 8.720, Y -21.020, Z 104.550}
   LaserEnd_Ext()
   LIN {X 8.720, Y -14.291, Z 104.550}
   LaserStart_Ext()
   LIN {X 8.720, Y 13.758, Z 104.550}
   LaserEnd_Ext()
   LIN {X 9.720, Y 9.705, Z 104.550}
   LaserStart_Ext()
   LIN {X 9.720, Y -16.758, Z 104.550}
   LaserEnd_Ext()
   LIN {X 9.720, Y -18.495, Z 104.550}
   LaserStart_Ext()
   LIN {X 9.720, Y -22.892, Z 104.550}
   LaserEnd_Ext()
   LIN {X 10.720, Y -21.410, Z 104.550}
   LaserStart_Ext()
   LIN {X 10.720, Y 3.790, Z 104.550}
   LaserEnd_Ext()
   LIN {X 11.720, Y -4.426, Z 104.550}
   LaserStart_Ext()
   LIN {X 11.720, Y -18.663, Z 104.550}
   LaserEnd_Ext()
   LIN {X 3.282, Y -12.685, Z 105.400}
   LaserStart_Ext()
   LIN {X 4.984, Y -12.657, Z 105.400} C_DIS
   LIN {X 6.247, Y -13.216, Z 105.400} C_DIS
   LIN {X 6.929, Y -13.515, Z 105.400} C_DIS
   LIN {X 7.635, Y -14.379, Z 105.400} C_DIS
   LIN {X 8.534, Y -15.486, Z 105.400} C_DIS
   LIN {X 8.764, Y -16.633, Z 105.400} C_DIS
   LIN {X 8.972, Y -17.652, Z 105.400} C_DIS
   LIN {X 8.597, Y -19.071, Z 105.400} C_DIS
   LIN {X 8.373, Y -19.913, Z 105.400} C_DIS
   LIN {X 7.927, Y -20.444, Z 105.400} C_DIS
   LIN {X 7.011, Y -21.529, Z 105.400} C_DIS
   LIN {X 6.135, Y -21.938, Z 105.400} C_DIS
   LIN {X 5.029, Y -22.457, Z 105.400} C_DIS
   LIN {X 3.295, Y -22.480, Z 105.400} C_DIS
   LIN {X 2.939, Y -22.486, Z 105.400} C_DIS
   LIN {X 2.713, Y -22.388, Z 105.400} C_DIS
   LIN {X 1.044, Y -21.659, Z 105.400} C_DIS
   LIN {X -0.186, Y -20.319, Z 105.400} C_DIS
   LIN {X -0.364, Y -20.124, Z 105.400} C_DIS
   LIN {X -0.452, Y -19.850, Z 105.400} C_DIS
   LIN {X -1.011, Y -18.140, Z 105.400} C_DIS
   LIN {X -0.468, Y -15.566, Z 105.400} C_DIS
   LIN {X -0.369, Y -15.102, Z 105.400} C_DIS
   LIN {X -0.183, Y -14.894, Z 105.400} C_DIS
   LIN {X 1.003, Y -13.553, Z 105.400} C_DIS
   LIN {X 2.611, Y -12.817, Z 105.400} C_DIS
   LIN {X 2.885, Y -12.691, Z 105.400} C_DIS
   LIN {X 3.282, Y -12.685, Z 105.400}
   LaserEnd_Ext()
   LIN {X -2.275, Y -4.343, Z 105.400}
   LaserStart_Ext()
   LIN {X -2.826, Y -7.788, Z 105.400} C_DIS
   LIN {X -3.315, Y -9.931, Z 105.400} C_DIS
   LIN {X -3.650, Y -11.408, Z 105.400} C_DIS
   LIN {X -4.043, Y -12.807, Z 105.400} C_DIS
   LIN {X -4.654, Y -14.960, Z 105.400} C_DIS
   LIN {X -4.975, Y -17.524, Z 105.400} C_DIS
   LIN {X -5.045, Y -18.107, Z 105.400} C_DIS
   LIN {X -4.900, Y -18.644, Z 105.400} C_DIS
   LIN {X -4.093, Y -21.693, Z 105.400} C_DIS
   LIN {X -2.683, Y -23.618, Z 105.400} C_DIS
   LIN {X -2.291, Y -24.115, Z 105.400} C_DIS
   LIN {X -1.111, Y -24.802, Z 105.400} C_DIS
   LIN {X 1.146, Y -26.164, Z 105.400} C_DIS
   LIN {X 6.713, Y -25.841, Z 105.400} C_DIS
   LIN {X 7.600, Y -25.800, Z 105.400} C_DIS
   LIN {X 7.923, Y -25.583, Z 105.400} C_DIS
   LIN {X 10.194, Y -24.045, Z 105.400} C_DIS
   LIN {X 10.718, Y -23.269, Z 105.400} C_DIS
   LIN {X 12.344, Y -20.829, Z 105.400} C_DIS
   LIN {X 12.888, Y -18.309, Z 105.400} C_DIS
   LIN {X 12.967, Y -17.934, Z 105.400} C_DIS
   LIN {X 12.989, Y -17.219, Z 105.400} C_DIS
   LIN {X 13.073, Y -14.674, Z 105.400} C_DIS
   LIN {X 13.083, Y -13.292, Z 105.400} C_DIS
   LIN {X 13.086, Y -11.714, Z 105.400} C_DIS
   LIN {X 12.997, Y -8.233, Z 105.400} C_DIS
   LIN {X 12.986, Y -7.911, Z 105.400} C_DIS
   LIN {X 12.801, Y -4.723, Z 105.400} C_DIS
   LIN {X 12.784, Y -4.516, Z 105.400} C_DIS
   LIN {X 12.317, Y 0.367, Z 105.400} C_DIS
   LIN {X 11.025, Y 8.402, Z 105.400} C_DIS
   LIN {X 10.917, Y 9.113, Z 105.400} C_DIS
   LIN {X 10.822, Y 9.519, Z 105.400} C_DIS
   LIN {X 8.669, Y 18.280, Z 105.400} C_DIS
   LIN {X 7.781, Y 20.986, Z 105.400} C_DIS
   LIN {X 6.452, Y 25.042, Z 105.400} C_DIS
   LIN {X 5.521, Y 27.353, Z 105.400} C_DIS
   LIN {X 3.422, Y 32.513, Z 105.400} C_DIS
   LIN {X 2.986, Y 33.443, Z 105.400} C_DIS
   LIN {X 1.119, Y 37.345, Z 105.400} C_DIS
   LIN {X 0.294, Y 38.927, Z 105.400} C_DIS
   LIN {X -0.843, Y 41.047, Z 105.400} C_DIS
   LIN {X -1.208, Y 41.700, Z 105.400} C_DIS
   LIN {X -2.235, Y 43.478, Z 105.400} C_DIS
   LIN {X -2.460, Y 43.870, Z 105.400} C_DIS
   LIN {X -2.538, Y 44.001, Z 105.400} C_DIS
   LIN {X -3.225, Y 45.139, Z 105.400} C_DIS
   LIN {X -4.115, Y 46.128, Z 105.400} C_DIS
   LIN {X -4.209, Y 46.232, Z 105.400} C_DIS
   LIN {X -4.405, Y 46.323, Z 105.400} C_DIS
   LIN {X -5.787, Y 46.964, Z 105.400} C_DIS
   LIN {X -6.804, Y 46.960, Z 105.400} C_DIS
   LIN {X -7.532, Y 46.956, Z 105.400} C_DIS
   LIN {X -8.195, Y 46.553, Z 105.400} C_DIS
   LIN {X -9.658, Y 45.667, Z 105.400} C_DIS
   LIN {X -10.295, Y 44.453, Z 105.400} C_DIS
   LIN {X -10.482, Y 44.097, Z 105.400} C_DIS
   LIN {X -10.506, Y 43.662, Z 105.400} C_DIS
   LIN {X -10.570, Y 42.497, Z 105.400} C_DIS
   LIN {X -10.196, Y 41.390, Z 105.400} C_DIS
   LIN {X -10.127, Y 41.186, Z 105.400} C_DIS
   LIN {X -10.026, Y 40.991, Z 105.400} C_DIS
   LIN {X -9.552, Y 40.075, Z 105.400} C_DIS
   LIN {X -9.210, Y 39.398, Z 105.400} C_DIS
   LIN {X -8.834, Y 38.646, Z 105.400} C_DIS
   LIN {X -8.415, Y 37.750, Z 105.400} C_DIS
   LIN {X -7.072, Y 34.727, Z 105.400} C_DIS
   LIN {X -6.421, Y 33.122, Z 105.400} C_DIS
   LIN {X -4.693, Y 28.084, Z 105.400} C_DIS
   LIN {X -4.123, Y 26.266, Z 105.400} C_DIS
   LIN {X -2.914, Y 20.982, Z 105.400} C_DIS
   LIN {X -2.216, Y 17.441, Z 105.400} C_DIS
   LIN {X -1.658, Y 11.393, Z 105.400} C_DIS
   LIN {X -1.403, Y 7.684, Z 105.400} C_DIS
   LIN {X -1.737, Y 1.742, Z 105.400} C_DIS
   LIN {X -1.860, Y -1.593, Z 105.400} C_DIS
   LIN {X -2.275, Y -4.343, Z 105.400}
   LaserEnd_Ext()
   LIN {X 7.945, Y -24.360, Z 105.400}
   LaserStart_Ext()
   LIN {X 0.093, Y -24.360, Z 105.400}
   LaserEnd_Ext()
   LIN {X -1.600, Y -23.360, Z 105.400}
   LaserStart_Ext()
   LIN {X 2.442, Y -23.360, Z 105.400}
   LaserEnd_Ext()
   LIN {X 5.459, Y -23.360, Z 105.400}
   LaserStart_Ext()
   LIN {X 9.421, Y -23.360, Z 105.400}
   LaserEnd_Ext()
   LIN {X 10.122, Y -22.360, Z 105.400}
   LaserStart_Ext()
   LIN {X 7.565, Y -22.360, Z 105.400}
   LaserEnd_Ext()
   LIN {X 0.333, Y -22.360, Z 105.400}
   LaserStart_Ext()
   LIN {X -2.364, Y -22.360, Z 105.400}
   LaserEnd_Ext()
   LIN {X -3.097, Y -21.360, Z 105.400}
   LaserStart_Ext()
   LIN {X -0.588, Y -21.360, Z 105.400}
   LaserEnd_Ext()
   LIN {X 8.462, Y -21.360, Z 105.400}
   LaserStart_Ext()
   LIN {X 10.788, Y -21.360, Z 105.400}
   LaserEnd_Ext()
   LIN {X 11.422, Y -20.360, Z 105.400}
   LaserStart_Ext()
   LIN {X 9.267, Y -20.360, Z 105.400}
   LaserEnd_Ext()
   LIN {X -1.339, Y -20.360, Z 105.400}
   LaserStart_Ext()
   LIN {X -3.411, Y -20.360, Z 105.400}
   LaserEnd_Ext()
   LIN {X -3.676, Y -19.360, Z 105.400}
   LaserStart_Ext()
   LIN {X -1.664, Y -19.360, Z 105.400}
   LaserEnd_Ext()
   LIN {X 9.555, Y -19.360, Z 105.400}
   LaserStart_Ext()
   LIN {X 11.638, Y -19.360, Z 105.400}
   LaserEnd_Ext()
   LIN {X 11.854, Y -18.360, Z 105.400}
   LaserStart_Ext()
   LIN {X 9.819, Y -18.360, Z 105.400}
   LaserEnd_Ext()
   LIN {X -1.986, Y -18.360, Z 105.400}
   LaserStart_Ext()
   LIN {X -3.941, Y -18.360, Z 105.400}
   LaserEnd_Ext()
   LIN {X -3.947, Y -17.360, Z 105.400}
   LaserStart_Ext()
   LIN {X -1.868, Y -17.360, Z 105.400}
   LaserEnd_Ext()
   LIN {X 9.933, Y -17.360, Z 105.400}
   LaserStart_Ext()
   LIN {X 11.984, Y -17.360, Z 105.400}
   LaserEnd_Ext()
   LIN {X 12.016, Y -16.360, Z 105.400}
   LaserStart_Ext()
   LIN {X 9.730, Y -16.360, Z 105.400}
   LaserEnd_Ext()
   LIN {X -1.658, Y -16.360, Z 105.400}
   LaserStart_Ext()
   LIN {X -3.821, Y -16.360, Z 105.400}
   LaserEnd_Ext()
   LIN {X -3.696, Y -15.360, Z 105.400}
   LaserStart_Ext()
   LIN {X -1.447, Y -15.360, Z 105.400}
   LaserEnd_Ext()
   LIN {X 9.529, Y -15.360, Z 105.400}
   LaserStart_Ext()
   LIN {X 12.049, Y -15.360, Z 105.400}
   LaserEnd_Ext()
   LIN {X 12.075, Y -14.360, Z 105.400}
   LaserStart_Ext()
   LIN {X 8.908, Y -14.360, Z 105.400}
   LaserEnd_Ext()
   LIN {X -1.047, Y -14.360, Z 105.400}
   LaserStart_Ext()
   LIN {X -3.444, Y -14.360, Z 105.400}
   LaserEnd_Ext()
   LIN {X -3.161, Y -13.360, Z 105.400}
   LaserStart_Ext()
   LIN {X -0.161, Y -13.360, Z 105.400}
   LaserEnd_Ext()
   LIN {X 8.094, Y -13.360, Z 105.400}
   LaserStart_Ext()
   LIN {X 12.082, Y -13.360, Z 105.400}
   LaserEnd_Ext()
   LIN {X 12.085, Y -12.360, Z 105.400}
   LaserStart_Ext()
   LIN {X 6.786, Y -12.360, Z 105.400}
   LaserEnd_Ext()
   LIN {X 1.207, Y -12.360, Z 105.400}
   LaserStart_Ext()
   LIN {X -2.879, Y -12.360, Z 105.400}
   LaserEnd_Ext()
   LIN {X -2.614, Y -11.360, Z 105.400}
   LaserStart_Ext()
   LIN {X 12.077, Y -11.360, Z 105.400}
   LaserEnd_Ext()
   LIN {X 12.051, Y -10.360, Z 105.400}
   LaserStart_Ext()
   LIN {X -2.387, Y -10.360, Z 105.400}
   LaserEnd_Ext()
   LIN {X -2.159, Y -9.360, Z 105.400}
   LaserStart_Ext()
   LIN {X 12.025, Y -9.360, Z 105.400}
   LaserEnd_Ext()
   LIN {X 11.999, Y -8.360, Z 105.400}
   LaserStart_Ext()
   LIN {X -1.931, Y -8.360, Z 105.400}
   LaserEnd_Ext()
   LIN {X -1.745, Y -7.360, Z 105.400}
   LaserStart_Ext()
   LIN {X 11.952, Y -7.360, Z 105.400}
   LaserEnd_Ext()
   LIN {X 11.894, Y -6.360, Z 105.400}
   LaserStart_Ext()
   LIN {X -1.585, Y -6.360, Z 105.400}
   LaserEnd_Ext()
   LIN {X -1.425, Y -5.360, Z 105.400}
   LaserStart_Ext()
   LIN {X 11.836, Y -5.360, Z 105.400}
   LaserEnd_Ext()
   LIN {X 11.764, Y -4.360, Z 105.400}
   LaserStart_Ext()
   LIN {X -1.266, Y -4.360, Z 105.400}
   LaserEnd_Ext()
   LIN {X -1.115, Y -3.360, Z 105.400}
   LaserStart_Ext()
   LIN {X 11.669, Y -3.360, Z 105.400}
   LaserEnd_Ext()
   LIN {X 11.573, Y -2.360, Z 105.400}
   LaserStart_Ext()
   LIN {X -0.965, Y -2.360, Z 105.400}
   LaserEnd_Ext()
   LIN {X -0.851, Y -1.360, Z 105.400}
   LaserStart_Ext()
   LIN {X 11.478, Y -1.360, Z 105.400}
   LaserEnd_Ext()
   LIN {X 11.382, Y -0.360, Z 105.400}
   LaserStart_Ext()
   LIN {X -0.814, Y -0.360, Z 105.400}
   LaserEnd_Ext()
   LIN {X -0.777, Y 0.640, Z 105.400}
   LaserStart_Ext()
   LIN {X 11.260, Y 0.640, Z 105.400}
   LaserEnd_Ext()
   LIN {X 11.100, Y 1.640, Z 105.400}
   LaserStart_Ext()
   LIN {X -0.740, Y 1.640, Z 105.400}
   LaserEnd_Ext()
   LIN {X -0.685, Y 2.640, Z 105.400}
   LaserStart_Ext()
   LIN {X 10.939, Y 2.640, Z 105.400}
   LaserEnd_Ext()
   LIN {X 10.778, Y 3.640, Z 105.400}
   LaserStart_Ext()
   LIN {X -0.629, Y 3.640, Z 105.400}
   LaserEnd_Ext()
   LIN {X -0.572, Y 4.640, Z 105.400}
   LaserStart_Ext()
   LIN {X 10.617, Y 4.640, Z 105.400}
   LaserEnd_Ext()
   LIN {X 10.456, Y 5.640, Z 105.400}
   LaserStart_Ext()
   LIN {X -0.516, Y 5.640, Z 105.400}
   LaserEnd_Ext()
   LIN {X -0.460, Y 6.640, Z 105.400}
   LaserStart_Ext()
   LIN {X 10.295, Y 6.640, Z 105.400}
   LaserEnd_Ext()
   LIN {X 10.134, Y 7.640, Z 105.400}
   LaserStart_Ext()
   LIN {X -0.405, Y 7.640, Z 105.400}
   LaserEnd_Ext()
   LIN {X -0.466, Y 8.640, Z 105.400}
   LaserStart_Ext()
   LIN {X 9.977, Y 8.640, Z 105.400}
   LaserEnd_Ext()
   LIN {X 9.763, Y 9.640, Z 105.400}
   LaserStart_Ext()
   LIN {X -0.535, Y 9.640, Z 105.400}
   LaserEnd_Ext()
   LIN {X -0.604, Y 10.640, Z 105.400}
   LaserStart_Ext()
   LIN {X 9.517, Y 10.640, Z 105.400}
   LaserEnd_Ext()
   LIN {X 9.271, Y 11.640, Z 105.400}
   LaserStart_Ext()
   LIN {X -0.677, Y 11.640, Z 105.400}
   LaserEnd_Ext()
   LIN {X -0.769, Y 12.640, Z 105.400}
   LaserStart_Ext()
   LIN {X 9.026, Y 12.640, Z 105.400}
   LaserEnd_Ext()
   LIN {X 8.780, Y 13.640, Z 105.400}
   LaserStart_Ext()
   LIN {X -0.861, Y 13.640, Z 105.400}
   LaserEnd_Ext()
   LIN {X -0.953, Y 14.640, Z 105.400}
   LaserStart_Ext()
   LIN {X 8.534, Y 14.640, Z 105.400}
   LaserEnd_Ext()
   LIN {X 8.288, Y 15.640, Z 105.400}
   LaserStart_Ext()
   LIN {X -1.045, Y 15.640, Z 105.400}
   LaserEnd_Ext()
   LIN {X -1.137, Y 16.640, Z 105.400}
   LaserStart_Ext()
   LIN {X 8.043, Y 16.640, Z 105.400}
   LaserEnd_Ext()
   LIN {X 7.797, Y 17.640, Z 105.400}
   LaserStart_Ext()
   LIN {X -1.235, Y 17.640, Z 105.400}
   LaserEnd_Ext()
   LIN {X -1.433, Y 18.640, Z 105.400}
   LaserStart_Ext()
   LIN {X 7.499, Y 18.640, Z 105.400}
   LaserEnd_Ext()
   LIN {X 7.171, Y 19.640, Z 105.400}
   LaserStart_Ext()
   LIN {X -1.630, Y 19.640, Z 105.400}
   LaserEnd_Ext()
   LIN {X -1.828, Y 20.640, Z 105.400}
   LaserStart_Ext()
   LIN {X 6.842, Y 20.640, Z 105.400}
   LaserEnd_Ext()
   LIN {X 6.515, Y 21.640, Z 105.400}
   LaserStart_Ext()
   LIN {X -2.039, Y 21.640, Z 105.400}
   LaserEnd_Ext()
   LIN {X -2.268, Y 22.640, Z 105.400}
   LaserStart_Ext()
   LIN {X 6.187, Y 22.640, Z 105.400}
   LaserEnd_Ext()
   LIN {X 5.859, Y 23.640, Z 105.400}
   LaserStart_Ext()
   LIN {X -2.497, Y 23.640, Z 105.400}
   LaserEnd_Ext()
   LIN {X -2.725, Y 24.640, Z 105.400}
   LaserStart_Ext()
   LIN {X 5.532, Y 24.640, Z 105.400}
   LaserEnd_Ext()
   LIN {X 5.133, Y 25.640, Z 105.400}
   LaserStart_Ext()
   LIN {X -2.954, Y 25.640, Z 105.400}
   LaserEnd_Ext()
   LIN {X -3.192, Y 26.640, Z 105.400}
   LaserStart_Ext()
   LIN {X 4.730, Y 26.640, Z 105.400}
   LaserEnd_Ext()
   LIN {X 4.324, Y 27.640, Z 105.400}
   LaserStart_Ext()
   LIN {X -3.506, Y 27.640, Z 105.400}
   LaserEnd_Ext()
   LIN {X -3.826, Y 28.640, Z 105.400}
   LaserStart_Ext()
   LIN {X 3.917, Y 28.640, Z 105.400}
   LaserEnd_Ext()
   LIN {X 3.511, Y 29.640, Z 105.400}
   LaserStart_Ext()
   LIN {X -4.169, Y 29.640, Z 105.400}
   LaserEnd_Ext()
   LIN {X -4.512, Y 30.640, Z 105.400}
   LaserStart_Ext()
   LIN {X 3.104, Y 30.640, Z 105.400}
   LaserEnd_Ext()
   LIN {X 2.697, Y 31.640, Z 105.400}
   LaserStart_Ext()
   LIN {X -4.855, Y 31.640, Z 105.400}
   LaserEnd_Ext()
   LIN {X -5.198, Y 32.640, Z 105.400}
   LaserStart_Ext()
   LIN {X 2.258, Y 32.640, Z 105.400}
   LaserEnd_Ext()
   LIN {X 1.783, Y 33.640, Z 105.400}
   LaserStart_Ext()
   LIN {X -5.552, Y 33.640, Z 105.400}
   LaserEnd_Ext()
   LIN {X -5.957, Y 34.640, Z 105.400}
   LaserStart_Ext()
   LIN {X 1.304, Y 34.640, Z 105.400}
   LaserEnd_Ext()
   LIN {X 0.826, Y 35.640, Z 105.400}
   LaserStart_Ext()
   LIN {X -6.383, Y 35.640, Z 105.400}
   LaserEnd_Ext()
   LIN {X -6.827, Y 36.640, Z 105.400}
   LaserStart_Ext()
   LIN {X 0.347, Y 36.640, Z 105.400}
   LaserEnd_Ext()
   LIN {X -0.163, Y 37.640, Z 105.400}
   LaserStart_Ext()
   LIN {X -7.271, Y 37.640, Z 105.400}
   LaserEnd_Ext()
   LIN {X -7.727, Y 38.640, Z 105.400}
   LaserStart_Ext()
   LIN {X -0.686, Y 38.640, Z 105.400}
   LaserEnd_Ext()
   LIN {X -1.223, Y 39.640, Z 105.400}
   LaserStart_Ext()
   LIN {X -8.213, Y 39.640, Z 105.400}
   LaserEnd_Ext()
   LIN {X -8.718, Y 40.640, Z 105.400}
   LaserStart_Ext()
   LIN {X -1.761, Y 40.640, Z 105.400}
   LaserEnd_Ext()
   LIN {X -2.328, Y 41.640, Z 105.400}
   LaserStart_Ext()
   LIN {X -9.225, Y 41.640, Z 105.400}
   LaserEnd_Ext()
   LIN {X -9.561, Y 42.640, Z 105.400}
   LaserStart_Ext()
   LIN {X -2.905, Y 42.640, Z 105.400}
   LaserEnd_Ext()
   LIN {X -3.488, Y 43.640, Z 105.400}
   LaserStart_Ext()
   LIN {X -9.506, Y 43.640, Z 105.400}
   LaserEnd_Ext()
   LIN {X -9.068, Y 44.640, Z 105.400}
   LaserStart_Ext()
   LIN {X -4.121, Y 44.640, Z 105.400}
   LaserEnd_Ext()
   LIN {X -5.309, Y 45.640, Z 105.400}
   LaserStart_Ext()
   LIN {X -7.772, Y 45.640, Z 105.400}
   LaserEnd_Ext()
   LIN {X 4.988, Y -12.596, Z 106.250}
   LaserStart_Ext()
   LIN {X 5.100, Y -12.616, Z 106.250} C_DIS
   LIN {X 6.999, Y -13.448, Z 106.250} C_DIS
   LIN {X 8.289, Y -15.027, Z 106.250} C_DIS
   LIN {X 8.609, Y -15.416, Z 106.250} C_DIS
   LIN {X 8.695, Y -15.831, Z 106.250} C_DIS
   LIN {X 9.052, Y -17.581, Z 106.250} C_DIS
   LIN {X 8.658, Y -19.072, Z 106.250} C_DIS
   LIN {X 8.455, Y -19.851, Z 106.250} C_DIS
   LIN {X 7.938, Y -20.460, Z 106.250} C_DIS
   LIN {X 7.078, Y -21.479, Z 106.250} C_DIS
   LIN {X 5.180, Y -22.365, Z 106.250} C_DIS
   LIN {X 5.062, Y -22.399, Z 106.250} C_DIS
   LIN {X 3.030, Y -22.428, Z 106.250} C_DIS
   LIN {X 1.664, Y -21.838, Z 106.250} C_DIS
   LIN {X 1.133, Y -21.606, Z 106.250} C_DIS
   LIN {X 0.614, Y -21.041, Z 106.250} C_DIS
   LIN {X -0.279, Y -20.074, Z 106.250} C_DIS
   LIN {X -0.692, Y -18.820, Z 106.250} C_DIS
   LIN {X -0.930, Y -18.092, Z 106.250} C_DIS
   LIN {X -0.690, Y -16.953, Z 106.250} C_DIS
   LIN {X -0.308, Y -15.074, Z 106.250} C_DIS
   LIN {X 0.527, Y -14.112, Z 106.250} C_DIS
   LIN {X 1.058, Y -13.512, Z 106.250} C_DIS
   LIN {X 1.589, Y -13.269, Z 106.250} C_DIS
   LIN {X 2.975, Y -12.629, Z 106.250} C_DIS
   LIN {X 4.988, Y -12.596, Z 106.250}
   LaserEnd_Ext()
   LIN {X -3.290, Y 45.182, Z 106.250}
   LaserStart_Ext()
   LIN {X -4.277, Y 46.273, Z 106.250} C_DIS
   LIN {X -5.498, Y 46.837, Z 106.250} C_DIS
   LIN {X -5.856, Y 47.001, Z 106.250} C_DIS
   LIN {X -6.486, Y 46.996, Z 106.250} C_DIS
   LIN {X -7.600, Y 46.988, Z 106.250} C_DIS
   LIN {X -9.529, Y 45.816, Z 106.250} C_DIS
   LIN {X -9.717, Y 45.702, Z 106.250} C_DIS
   LIN {X -9.854, Y 45.442, Z 106.250} C_DIS
   LIN {X -10.541, Y 44.133, Z 106.250} C_DIS
   LIN {X -10.624, Y 42.655, Z 106.250} C_DIS
   LIN {X -10.630, Y 42.538, Z 106.250} C_DIS
   LIN {X -10.182, Y 41.212, Z 106.250} C_DIS
   LIN {X -9.806, Y 40.494, Z 106.250} C_DIS
   LIN {X -9.604, Y 40.104, Z 106.250} C_DIS
   LIN {X -9.175, Y 39.254, Z 106.250} C_DIS
   LIN {X -8.883, Y 38.676, Z 106.250} C_DIS
   LIN {X -8.715, Y 38.319, Z 106.250} C_DIS
   LIN {X -8.164, Y 37.142, Z 106.250} C_DIS
   LIN {X -7.210, Y 34.993, Z 106.250} C_DIS
   LIN {X -6.292, Y 32.731, Z 106.250} C_DIS
   LIN {X -4.878, Y 28.608, Z 106.250} C_DIS
   LIN {X -4.040, Y 25.932, Z 106.250} C_DIS
   LIN {X -2.992, Y 21.350, Z 106.250} C_DIS
   LIN {X -2.171, Y 17.192, Z 106.250} C_DIS
   LIN {X -1.682, Y 11.887, Z 106.250} C_DIS
   LIN {X -1.376, Y 7.434, Z 106.250} C_DIS
   LIN {X -1.776, Y 0.299, Z 106.250} C_DIS
   LIN {X -1.858, Y -1.914, Z 106.250} C_DIS
   LIN {X -2.133, Y -3.739, Z 106.250} C_DIS
   LIN {X -2.792, Y -7.855, Z 106.250} C_DIS
   LIN {X -3.025, Y -8.878, Z 106.250} C_DIS
   LIN {X -3.635, Y -11.564, Z 106.250} C_DIS
   LIN {X -4.350, Y -14.108, Z 106.250} C_DIS
   LIN {X -4.580, Y -14.920, Z 106.250} C_DIS
   LIN {X -4.701, Y -15.888, Z 106.250} C_DIS
   LIN {X -4.965, Y -18.068, Z 106.250} C_DIS
   LIN {X -4.422, Y -20.075, Z 106.250} C_DIS
   LIN {X -4.004, Y -21.652, Z 106.250} C_DIS
   LIN {X -3.275, Y -22.647, Z 106.250} C_DIS
   LIN {X -2.063, Y -24.185, Z 106.250} C_DIS
   LIN {X 1.182, Y -26.073, Z 106.250} C_DIS
   LIN {X 1.285, Y -26.124, Z 106.250} C_DIS
   LIN {X 1.438, Y -26.134, Z 106.250} C_DIS
   LIN {X 7.298, Y -25.850, Z 106.250} C_DIS
   LIN {X 7.681, Y -25.740, Z 106.250} C_DIS
   LIN {X 10.097, Y -24.102, Z 106.250} C_DIS
   LIN {X 10.350, Y -23.904, Z 106.250} C_DIS
   LIN {X 10.845, Y -23.130, Z 106.250} C_DIS
   LIN {X 12.431, Y -20.750, Z 106.250} C_DIS
   LIN {X 12.714, Y -19.439, Z 106.250} C_DIS
   LIN {X 13.049, Y -17.854, Z 106.250} C_DIS
   LIN {X 13.138, Y -14.826, Z 106.250} C_DIS
   LIN {X 13.146, Y -14.594, Z 106.250} C_DIS
   LIN {X 13.147, Y -14.467, Z 106.250} C_DIS
   LIN {X 13.152, Y -11.633, Z 106.250} C_DIS
   LIN {X 13.096, Y -9.442, Z 106.250} C_DIS
   LIN {X 13.044, Y -7.830, Z 106.250} C_DIS
   LIN {X 12.902, Y -5.389, Z 106.250} C_DIS
   LIN {X 12.756, Y -3.632, Z 106.250} C_DIS
   LIN {X 12.408, Y 0.013, Z 106.250} C_DIS
   LIN {X 11.443, Y 6.011, Z 106.250} C_DIS
   LIN {X 11.036, Y 8.697, Z 106.250} C_DIS
   LIN {X 10.678, Y 10.231, Z 106.250} C_DIS
   LIN {X 8.759, Y 18.041, Z 106.250} C_DIS
   LIN {X 7.679, Y 21.331, Z 106.250} C_DIS
   LIN {X 6.503, Y 24.919, Z 106.250} C_DIS
   LIN {X 5.388, Y 27.686, Z 106.250} C_DIS
   LIN {X 3.543, Y 32.221, Z 106.250} C_DIS
   LIN {X 2.696, Y 34.027, Z 106.250} C_DIS
   LIN {X 1.277, Y 36.993, Z 106.250} C_DIS
   LIN {X 0.056, Y 39.336, Z 106.250} C_DIS
   LIN {X -0.525, Y 40.420, Z 106.250} C_DIS
   LIN {X -1.486, Y 42.138, Z 106.250} C_DIS
   LIN {X -1.807, Y 42.694, Z 106.250} C_DIS
   LIN {X -2.522, Y 43.914, Z 106.250} C_DIS
   LIN {X -3.279, Y 45.163, Z 106.250}
   LaserEnd_Ext()
   LIN {X 11.602, Y -19.852, Z 106.250}
   LaserStart_Ext()
   LIN {X 11.602, Y -2.068, Z 106.250}
   LaserEnd_Ext()
   LIN {X 10.602, Y 4.943, Z 106.250}
   LaserStart_Ext()
   LIN {X 10.602, Y -21.691, Z 106.250}
   LaserEnd_Ext()
   LIN {X 9.602, Y -23.217, Z 106.250}
   LaserStart_Ext()
   LIN {X 9.602, Y -19.415, Z 106.250}
   LaserEnd_Ext()
   LIN {X 9.602, Y -15.278, Z 106.250}
   LaserStart_Ext()
   LIN {X 9.602, Y 10.420, Z 106.250}
   LaserEnd_Ext()
   LIN {X 8.602, Y 14.489, Z 106.250}
   LaserStart_Ext()
   LIN {X 8.602, Y -13.829, Z 106.250}
   LaserEnd_Ext()
   LIN {X 8.602, Y -21.224, Z 106.250}
   LaserStart_Ext()
   LIN {X 8.602, Y -23.907, Z 106.250}
   LaserEnd_Ext()
   LIN {X 7.602, Y -24.585, Z 106.250}
   LaserStart_Ext()
   LIN {X 7.602, Y -22.331, Z 106.250}
   LaserEnd_Ext()
   LIN {X 7.602, Y -12.652, Z 106.250}
   LaserStart_Ext()
   LIN {X 7.602, Y 18.359, Z 106.250}
   LaserEnd_Ext()
   LIN {X 6.602, Y 21.407, Z 106.250}
   LaserStart_Ext()
   LIN {X 6.602, Y -12.182, Z 106.250}
   LaserEnd_Ext()
   LIN {X 6.602, Y -22.805, Z 106.250}
   LaserStart_Ext()
   LIN {X 6.602, Y -24.883, Z 106.250}
   LaserEnd_Ext()
   LIN {X 5.602, Y -24.931, Z 106.250}
   LaserStart_Ext()
   LIN {X 5.602, Y -23.272, Z 106.250}
   LaserEnd_Ext()
   LIN {X 5.602, Y -11.744, Z 106.250}
   LaserStart_Ext()
   LIN {X 5.602, Y 24.458, Z 106.250}
   LaserEnd_Ext()
   LIN {X 4.602, Y 26.961, Z 106.250}
   LaserStart_Ext()
   LIN {X 4.602, Y -11.602, Z 106.250}
   LaserEnd_Ext()
   LIN {X 4.602, Y -23.405, Z 106.250}
   LaserStart_Ext()
   LIN {X 4.602, Y -24.980, Z 106.250}
   LaserEnd_Ext()
   LIN {X 3.602, Y -25.028, Z 106.250}
   LaserStart_Ext()
   LIN {X 3.602, Y -23.420, Z 106.250}
   LaserEnd_Ext()
   LIN {X 3.602, Y -11.619, Z 106.250}
   LaserStart_Ext()
   LIN {X 3.602, Y 29.422, Z 106.250}
   LaserEnd_Ext()
   LIN {X 2.602, Y 31.873, Z 106.250}
   LaserStart_Ext()
   LIN {X 2.602, Y -11.703, Z 106.250}
   LaserEnd_Ext()
   LIN {X 2.602, Y -23.333, Z 106.250}
   LaserStart_Ext()
   LIN {X 2.602, Y -25.077, Z 106.250}
   LaserEnd_Ext()
   LIN {X 1.602, Y -25.125, Z 106.250}
   LaserStart_Ext()
   LIN {X 1.602, Y -22.901, Z 106.250}
   LaserEnd_Ext()
   LIN {X 1.602, Y -12.161, Z 106.250}
   LaserStart_Ext()
   LIN {X 1.602, Y 33.998, Z 106.250}
   LaserEnd_Ext()
   LIN {X 0.602, Y 36.087, Z 106.250}
   LaserStart_Ext()
   LIN {X 0.602, Y -12.623, Z 106.250}
   LaserEnd_Ext()
   LIN {X 0.602, Y -22.452, Z 106.250}
   LaserStart_Ext()
   LIN {X 0.602, Y -24.578, Z 106.250}
   LaserEnd_Ext()
   LIN {X -0.398, Y -23.997, Z 106.250}
   LaserStart_Ext()
   LIN {X -0.398, Y -21.419, Z 106.250}
   LaserEnd_Ext()
   LIN {X -0.398, Y -13.653, Z 106.250}
   LaserStart_Ext()
   LIN {X -0.398, Y 7.006, Z 106.250}
   LaserEnd_Ext()
   LIN {X -0.398, Y 7.794, Z 106.250}
   LaserStart_Ext()
   LIN {X -0.398, Y 38.044, Z 106.250}
   LaserEnd_Ext()
   LIN {X -1.398, Y 39.932, Z 106.250}
   LaserStart_Ext()
   LIN {X -1.398, Y 18.441, Z 106.250}
   LaserEnd_Ext()
   LIN {X -1.398, Y -5.474, Z 106.250}
   LaserStart_Ext()
   LIN {X -1.398, Y -15.418, Z 106.250}
   LaserEnd_Ext()
   LIN {X -1.398, Y -19.873, Z 106.250}
   LaserStart_Ext()
   LIN {X -1.398, Y -23.413, Z 106.250}
   LaserEnd_Ext()
   LIN {X -2.398, Y -22.144, Z 106.250}
   LaserStart_Ext()
   LIN {X -2.398, Y -10.634, Z 106.250}
   LaserEnd_Ext()
   LIN {X -2.398, Y 23.240, Z 106.250}
   LaserStart_Ext()
   LIN {X -2.398, Y 41.718, Z 106.250}
   LaserEnd_Ext()
   LIN {X -3.398, Y 43.431, Z 106.250}
   LaserStart_Ext()
   LIN {X -3.398, Y 27.229, Z 106.250}
   LaserEnd_Ext()
   LIN {X -3.398, Y -14.418, Z 106.250}
   LaserStart_Ext()
   LIN {X -3.398, Y -20.034, Z 106.250}
   LaserEnd_Ext()
   LIN {X -4.398, Y 30.291, Z 106.250}
   LaserStart_Ext()
   LIN {X -4.398, Y 44.916, Z 106.250}
   LaserEnd_Ext()
   LIN {X -5.398, Y 45.689, Z 106.250}
   LaserStart_Ext()
   LIN {X -5.398, Y 33.187, Z 106.250}
   LaserEnd_Ext()
   LIN {X -6.398, Y 35.629, Z 106.250}
   LaserStart_Ext()
   LIN {X -6.398, Y 45.996, Z 106.250}
   LaserEnd_Ext()
   LIN {X -7.398, Y 45.941, Z 106.250}
   LaserStart_Ext()
   LIN {X -7.398, Y 37.864, Z 106.250}
   LaserEnd_Ext()
   LIN {X -8.398, Y 39.934, Z 106.250}
   LaserStart_Ext()
   LIN {X -8.398, Y 45.333, Z 106.250}
   LaserEnd_Ext()
   LIN {X -9.398, Y 44.159, Z 106.250}
   LaserStart_Ext()
   LIN {X -9.398, Y 42.016, Z 106.250}
   LaserEnd_Ext()
   LIN {X 5.121, Y -12.533, Z 107.100}
   LaserStart_Ext()
   LIN {X 6.816, Y -13.271, Z 107.100} C_DIS
   LIN {X 7.069, Y -13.382, Z 107.100} C_DIS
   LIN {X 7.232, Y -13.581, Z 107.100} C_DIS
   LIN {X 8.684, Y -15.346, Z 107.100} C_DIS
   LIN {X 9.073, Y -17.226, Z 107.100} C_DIS
   LIN {X 9.131, Y -17.510, Z 107.100} C_DIS
   LIN {X 9.067, Y -17.752, Z 107.100} C_DIS
   LIN {X 8.536, Y -19.788, Z 107.100} C_DIS
   LIN {X 7.186, Y -21.381, Z 107.100} C_DIS
   LIN {X 7.054, Y -21.472, Z 107.100} C_DIS
   LIN {X 5.189, Y -22.338, Z 107.100} C_DIS
   LIN {X 3.910, Y -22.359, Z 107.100} C_DIS
   LIN {X 3.120, Y -22.371, Z 107.100} C_DIS
   LIN {X 2.088, Y -21.925, Z 107.100} C_DIS
   LIN {X 1.222, Y -21.553, Z 107.100} C_DIS
   LIN {X 0.697, Y -20.988, Z 107.100} C_DIS
   LIN {X -0.194, Y -20.024, Z 107.100} C_DIS
   LIN {X -0.604, Y -18.778, Z 107.100} C_DIS
   LIN {X -0.849, Y -18.044, Z 107.100} C_DIS
   LIN {X -0.660, Y -17.069, Z 107.100} C_DIS
   LIN {X -0.250, Y -15.054, Z 107.100} C_DIS
   LIN {X 0.681, Y -13.981, Z 107.100} C_DIS
   LIN {X 1.123, Y -13.463, Z 107.100} C_DIS
   LIN {X 3.065, Y -12.567, Z 107.100} C_DIS
   LIN {X 5.121, Y -12.533, Z 107.100}
   LaserEnd_Ext()
   LIN {X 8.848, Y 17.801, Z 107.100}
   LaserStart_Ext()
   LIN {X 10.534, Y 10.943, Z 107.100} C_DIS
   LIN {X 11.155, Y 8.280, Z 107.100} C_DIS
   LIN {X 11.861, Y 3.619, Z 107.100} C_DIS
   LIN {X 12.498, Y -0.341, Z 107.100} C_DIS
   LIN {X 12.728, Y -2.748, Z 107.100} C_DIS
   LIN {X 13.004, Y -6.054, Z 107.100} C_DIS
   LIN {X 13.102, Y -7.749, Z 107.100} C_DIS
   LIN {X 13.196, Y -10.652, Z 107.100} C_DIS
   LIN {X 13.219, Y -11.553, Z 107.100} C_DIS
   LIN {X 13.216, Y -12.847, Z 107.100} C_DIS
   LIN {X 13.219, Y -14.513, Z 107.100} C_DIS
   LIN {X 13.194, Y -15.605, Z 107.100} C_DIS
   LIN {X 13.130, Y -17.773, Z 107.100} C_DIS
   LIN {X 12.540, Y -20.569, Z 107.100} C_DIS
   LIN {X 12.518, Y -20.672, Z 107.100} C_DIS
   LIN {X 12.394, Y -20.857, Z 107.100} C_DIS
   LIN {X 10.603, Y -23.657, Z 107.100} C_DIS
   LIN {X 9.688, Y -24.374, Z 107.100} C_DIS
   LIN {X 7.762, Y -25.679, Z 107.100} C_DIS
   LIN {X 6.619, Y -26.009, Z 107.100} C_DIS
   LIN {X 2.906, Y -26.189, Z 107.100} C_DIS
   LIN {X 1.470, Y -26.093, Z 107.100} C_DIS
   LIN {X 0.498, Y -25.612, Z 107.100} C_DIS
   LIN {X -1.836, Y -24.254, Z 107.100} C_DIS
   LIN {X -3.867, Y -21.676, Z 107.100} C_DIS
   LIN {X -3.943, Y -21.506, Z 107.100} C_DIS
   LIN {X -4.884, Y -18.029, Z 107.100} C_DIS
   LIN {X -4.568, Y -15.415, Z 107.100} C_DIS
   LIN {X -4.506, Y -14.881, Z 107.100} C_DIS
   LIN {X -4.341, Y -14.288, Z 107.100} C_DIS
   LIN {X -3.619, Y -11.720, Z 107.100} C_DIS
   LIN {X -2.806, Y -8.137, Z 107.100} C_DIS
   LIN {X -2.764, Y -7.957, Z 107.100} C_DIS
   LIN {X -2.686, Y -7.476, Z 107.100} C_DIS
   LIN {X -1.992, Y -3.135, Z 107.100} C_DIS
   LIN {X -1.856, Y -2.236, Z 107.100} C_DIS
   LIN {X -1.816, Y -1.145, Z 107.100} C_DIS
   LIN {X -1.348, Y 7.183, Z 107.100} C_DIS
   LIN {X -1.706, Y 12.381, Z 107.100} C_DIS
   LIN {X -2.126, Y 16.942, Z 107.100} C_DIS
   LIN {X -3.069, Y 21.719, Z 107.100} C_DIS
   LIN {X -3.956, Y 25.599, Z 107.100} C_DIS
   LIN {X -5.063, Y 29.132, Z 107.100} C_DIS
   LIN {X -6.164, Y 32.340, Z 107.100} C_DIS
   LIN {X -7.348, Y 35.259, Z 107.100} C_DIS
   LIN {X -7.914, Y 36.534, Z 107.100} C_DIS
   LIN {X -8.241, Y 37.232, Z 107.100} C_DIS
   LIN {X -8.932, Y 38.705, Z 107.100} C_DIS
   LIN {X -9.323, Y 39.478, Z 107.100} C_DIS
   LIN {X -9.657, Y 40.131, Z 107.100} C_DIS
   LIN {X -10.070, Y 40.919, Z 107.100} C_DIS
   LIN {X -10.237, Y 41.239, Z 107.100} C_DIS
   LIN {X -10.321, Y 41.485, Z 107.100} C_DIS
   LIN {X -10.695, Y 42.602, Z 107.100} C_DIS
   LIN {X -10.602, Y 44.139, Z 107.100} C_DIS
   LIN {X -9.775, Y 45.740, Z 107.100} C_DIS
   LIN {X -7.670, Y 47.020, Z 107.100} C_DIS
   LIN {X -6.937, Y 47.028, Z 107.100} C_DIS
   LIN {X -5.926, Y 47.037, Z 107.100} C_DIS
   LIN {X -4.512, Y 46.389, Z 107.100} C_DIS
   LIN {X -4.345, Y 46.313, Z 107.100} C_DIS
   LIN {X -4.267, Y 46.227, Z 107.100} C_DIS
   LIN {X -3.358, Y 45.224, Z 107.100} C_DIS
   LIN {X -2.675, Y 44.108, Z 107.100} C_DIS
   LIN {X -2.584, Y 43.959, Z 107.100} C_DIS
   LIN {X -2.424, Y 43.686, Z 107.100} C_DIS
   LIN {X -1.614, Y 42.307, Z 107.100} C_DIS
   LIN {X -0.208, Y 39.794, Z 107.100} C_DIS
   LIN {X 1.435, Y 36.642, Z 107.100} C_DIS
   LIN {X 2.407, Y 34.612, Z 107.100} C_DIS
   LIN {X 3.665, Y 31.929, Z 107.100} C_DIS
   LIN {X 5.255, Y 28.019, Z 107.100} C_DIS
   LIN {X 6.554, Y 24.796, Z 107.100} C_DIS
   LIN {X 7.577, Y 21.676, Z 107.100} C_DIS
   LIN {X 8.848, Y 17.801, Z 107.100}
   LaserEnd_Ext()
   LIN {X -8.209, Y 45.522, Z 107.100}
   LaserStart_Ext()
   LIN {X -5.019, Y 45.522, Z 107.100}
   LaserEnd_Ext()
   LIN {X -4.101, Y 44.522, Z 107.100}
   LaserStart_Ext()
   LIN {X -9.286, Y 44.522, Z 107.100}
   LaserEnd_Ext()
   LIN {X -9.637, Y 43.522, Z 107.100}
   LaserStart_Ext()
   LIN {X -3.488, Y 43.522, Z 107.100}
   LaserEnd_Ext()
   LIN {X -2.900, Y 42.522, Z 107.100}
   LaserStart_Ext()
   LIN {X -9.613, Y 42.522, Z 107.100}
   LaserEnd_Ext()
   LIN {X -9.257, Y 41.522, Z 107.100}
   LaserStart_Ext()
   LIN {X -2.320, Y 41.522, Z 107.100}
   LaserEnd_Ext()
   LIN {X -1.761, Y 40.522, Z 107.100}
   LaserStart_Ext()
   LIN {X -8.733, Y 40.522, Z 107.100}
   LaserEnd_Ext()
   LIN {X -8.225, Y 39.522, Z 107.100}
   LaserStart_Ext()
   LIN {X -1.201, Y 39.522, Z 107.100}
   LaserEnd_Ext()
   LIN {X -0.672, Y 38.522, Z 107.100}
   LaserStart_Ext()
   LIN {X -7.741, Y 38.522, Z 107.100}
   LaserEnd_Ext()
   LIN {X -7.272, Y 37.522, Z 107.100}
   LaserStart_Ext()
   LIN {X -0.151, Y 37.522, Z 107.100}
   LaserEnd_Ext()
   LIN {X 0.370, Y 36.522, Z 107.100}
   LaserStart_Ext()
   LIN {X -6.814, Y 36.522, Z 107.100}
   LaserEnd_Ext()
   LIN {X -6.375, Y 35.522, Z 107.100}
   LaserStart_Ext()
   LIN {X 0.863, Y 35.522, Z 107.100}
   LaserEnd_Ext()
   LIN {X 1.341, Y 34.522, Z 107.100}
   LaserStart_Ext()
   LIN {X -5.970, Y 34.522, Z 107.100}
   LaserEnd_Ext()
   LIN {X -5.564, Y 33.522, Z 107.100}
   LaserStart_Ext()
   LIN {X 1.813, Y 33.522, Z 107.100}
   LaserEnd_Ext()
   LIN {X 2.282, Y 32.522, Z 107.100}
   LaserStart_Ext()
   LIN {X -5.169, Y 32.522, Z 107.100}
   LaserEnd_Ext()
   LIN {X -4.826, Y 31.522, Z 107.100}
   LaserStart_Ext()
   LIN {X 2.751, Y 31.522, Z 107.100}
   LaserEnd_Ext()
   LIN {X 3.158, Y 30.522, Z 107.100}
   LaserStart_Ext()
   LIN {X -4.483, Y 30.522, Z 107.100}
   LaserEnd_Ext()
   LIN {X -4.140, Y 29.522, Z 107.100}
   LaserStart_Ext()
   LIN {X 3.564, Y 29.522, Z 107.100}
   LaserEnd_Ext()
   LIN {X 3.971, Y 28.522, Z 107.100}
   LaserStart_Ext()
   LIN {X -3.824, Y 28.522, Z 107.100}
   LaserEnd_Ext()
   LIN {X -3.511, Y 27.522, Z 107.100}
   LaserStart_Ext()
   LIN {X 4.377, Y 27.522, Z 107.100}
   LaserEnd_Ext()
   LIN {X 4.780, Y 26.522, Z 107.100}
   LaserStart_Ext()
   LIN {X -3.198, Y 26.522, Z 107.100}
   LaserEnd_Ext()
   LIN {X -2.913, Y 25.522, Z 107.100}
   LaserStart_Ext()
   LIN {X 5.184, Y 25.522, Z 107.100}
   LaserEnd_Ext()
   LIN {X 5.587, Y 24.522, Z 107.100}
   LaserStart_Ext()
   LIN {X -2.684, Y 24.522, Z 107.100}
   LaserEnd_Ext()
   LIN {X -2.456, Y 23.522, Z 107.100}
   LaserStart_Ext()
   LIN {X 5.920, Y 23.522, Z 107.100}
   LaserEnd_Ext()
   LIN {X 6.247, Y 22.522, Z 107.100}
   LaserStart_Ext()
   LIN {X -2.227, Y 22.522, Z 107.100}
   LaserEnd_Ext()
   LIN {X -2.011, Y 21.522, Z 107.100}
   LaserStart_Ext()
   LIN {X 6.575, Y 21.522, Z 107.100}
   LaserEnd_Ext()
   LIN {X 6.903, Y 20.522, Z 107.100}
   LaserStart_Ext()
   LIN {X -1.813, Y 20.522, Z 107.100}
   LaserEnd_Ext()
   LIN {X -1.616, Y 19.522, Z 107.100}
   LaserStart_Ext()
   LIN {X 7.231, Y 19.522, Z 107.100}
   LaserEnd_Ext()
   LIN {X 7.559, Y 18.522, Z 107.100}
   LaserStart_Ext()
   LIN {X -1.419, Y 18.522, Z 107.100}
   LaserEnd_Ext()
   LIN {X -1.221, Y 17.522, Z 107.100}
   LaserStart_Ext()
   LIN {X 7.887, Y 17.522, Z 107.100}
   LaserEnd_Ext()
   LIN {X 8.133, Y 16.522, Z 107.100}
   LaserStart_Ext()
   LIN {X -1.083, Y 16.522, Z 107.100}
   LaserEnd_Ext()
   LIN {X -0.991, Y 15.522, Z 107.100}
   LaserStart_Ext()
   LIN {X 8.379, Y 15.522, Z 107.100}
   LaserEnd_Ext()
   LIN {X 8.625, Y 14.522, Z 107.100}
   LaserStart_Ext()
   LIN {X -0.899, Y 14.522, Z 107.100}
   LaserEnd_Ext()
   LIN {X -0.807, Y 13.522, Z 107.100}
   LaserStart_Ext()
   LIN {X 8.870, Y 13.522, Z 107.100}
   LaserEnd_Ext()
   LIN {X 9.116, Y 12.522, Z 107.100}
   LaserStart_Ext()
   LIN {X -0.715, Y 12.522, Z 107.100}
   LaserEnd_Ext()
   LIN {X -0.644, Y 11.522, Z 107.100}
   LaserStart_Ext()
   LIN {X 9.362, Y 11.522, Z 107.100}
   LaserEnd_Ext()
   LIN {X 9.605, Y 10.522, Z 107.100}
   LaserStart_Ext()
   LIN {X -0.576, Y 10.522, Z 107.100}
   LaserEnd_Ext()
   LIN {X -0.507, Y 9.522, Z 107.100}
   LaserStart_Ext()
   LIN {X 9.838, Y 9.522, Z 107.100}
   LaserEnd_Ext()
   LIN {X 10.072, Y 8.522, Z 107.100}
   LaserStart_Ext()
   LIN {X -0.438, Y 8.522, Z 107.100}
   LaserEnd_Ext()
   LIN {X -0.369, Y 7.522, Z 107.100}
   LaserStart_Ext()
   LIN {X 10.258, Y 7.522, Z 107.100}
   LaserEnd_Ext()
   LIN {X 10.410, Y 6.522, Z 107.100}
   LaserStart_Ext()
   LIN {X -0.384, Y 6.522, Z 107.100}
   LaserEnd_Ext()
   LIN {X -0.440, Y 5.522, Z 107.100}
   LaserStart_Ext()
   LIN {X 10.561, Y 5.522, Z 107.100}
   LaserEnd_Ext()
   LIN {X 10.713, Y 4.522, Z 107.100}
   LaserStart_Ext()
   LIN {X -0.496, Y 4.522, Z 107.100}
   LaserEnd_Ext()
   LIN {X -0.552, Y 3.522, Z 107.100}
   LaserStart_Ext()
   LIN {X 10.865, Y 3.522, Z 107.100}
   LaserEnd_Ext()
   LIN {X 11.025, Y 2.522, Z 107.100}
   LaserStart_Ext()
   LIN {X -0.608, Y 2.522, Z 107.100}
   LaserEnd_Ext()
   LIN {X -0.665, Y 1.522, Z 107.100}
   LaserStart_Ext()
   LIN {X 11.186, Y 1.522, Z 107.100}
   LaserEnd_Ext()
   LIN {X 11.347, Y 0.522, Z 107.100}
   LaserStart_Ext()
   LIN {X -0.721, Y 0.522, Z 107.100}
   LaserEnd_Ext()
   LIN {X -0.777, Y -0.478, Z 107.100}
   LaserStart_Ext()
   LIN {X 11.507, Y -0.478, Z 107.100}
   LaserEnd_Ext()
   LIN {X 11.602, Y -1.478, Z 107.100}
   LaserStart_Ext()
   LIN {X -0.828, Y -1.478, Z 107.100}
   LaserEnd_Ext()
   LIN {X -0.882, Y -2.478, Z 107.100}
   LaserStart_Ext()
   LIN {X 11.698, Y -2.478, Z 107.100}
   LaserEnd_Ext()
   LIN {X 11.786, Y -3.478, Z 107.100}
   LaserStart_Ext()
   LIN {X -1.034, Y -3.478, Z 107.100}
   LaserEnd_Ext()
   LIN {X -1.194, Y -4.478, Z 107.100}
   LaserStart_Ext()
   LIN {X 11.869, Y -4.478, Z 107.100}
   LaserEnd_Ext()
   LIN {X 11.952, Y -5.478, Z 107.100}
   LaserStart_Ext()
   LIN {X -1.354, Y -5.478, Z 107.100}
   LaserEnd_Ext()
   LIN {X -1.514, Y -6.478, Z 107.100}
   LaserStart_Ext()
   LIN {X 12.027, Y -6.478, Z 107.100}
   LaserEnd_Ext()
   LIN {X 12.085, Y -7.478, Z 107.100}
   LaserStart_Ext()
   LIN {X -1.674, Y -7.478, Z 107.100}
   LaserEnd_Ext()
   LIN {X -1.858, Y -8.478, Z 107.100}
   LaserStart_Ext()
   LIN {X 12.125, Y -8.478, Z 107.100}
   LaserEnd_Ext()
   LIN {X 12.157, Y -9.478, Z 107.100}
   LaserStart_Ext()
   LIN {X -2.085, Y -9.478, Z 107.100}
   LaserEnd_Ext()
   LIN {X -2.312, Y -10.478, Z 107.100}
   LaserStart_Ext()
   LIN {X 12.190, Y -10.478, Z 107.100}
   LaserEnd_Ext()
   LIN {X 12.217, Y -11.478, Z 107.100}
   LaserStart_Ext()
   LIN {X -2.539, Y -11.478, Z 107.100}
   LaserEnd_Ext()
   LIN {X -2.794, Y -12.478, Z 107.100}
   LaserStart_Ext()
   LIN {X 0.870, Y -12.478, Z 107.100}
   LaserEnd_Ext()
   LIN {X 7.495, Y -12.478, Z 107.100}
   LaserStart_Ext()
   LIN {X 12.217, Y -12.478, Z 107.100}
   LaserEnd_Ext()
   LIN {X 12.217, Y -13.478, Z 107.100}
   LaserStart_Ext()
   LIN {X 8.442, Y -13.478, Z 107.100}
   LaserEnd_Ext()
   LIN {X -0.207, Y -13.478, Z 107.100}
   LaserStart_Ext()
   LIN {X -3.075, Y -13.478, Z 107.100}
   LaserEnd_Ext()
   LIN {X -3.356, Y -14.478, Z 107.100}
   LaserStart_Ext()
   LIN {X -1.068, Y -14.478, Z 107.100}
   LaserEnd_Ext()
   LIN {X 9.265, Y -14.478, Z 107.100}
   LaserStart_Ext()
   LIN {X 12.219, Y -14.478, Z 107.100}
   LaserEnd_Ext()
   LIN {X 12.196, Y -15.478, Z 107.100}
   LaserStart_Ext()
   LIN {X 9.733, Y -15.478, Z 107.100}
   LaserEnd_Ext()
   LIN {X -1.357, Y -15.478, Z 107.100}
   LaserStart_Ext()
   LIN {X -3.569, Y -15.478, Z 107.100}
   LaserEnd_Ext()
   LIN {X -3.689, Y -16.478, Z 107.100}
   LaserStart_Ext()
   LIN {X -1.561, Y -16.478, Z 107.100}
   LaserEnd_Ext()
   LIN {X 9.940, Y -16.478, Z 107.100}
   LaserStart_Ext()
   LIN {X 12.168, Y -16.478, Z 107.100}
   LaserEnd_Ext()
   LIN {X 12.138, Y -17.478, Z 107.100}
   LaserStart_Ext()
   LIN {X 10.130, Y -17.478, Z 107.100}
   LaserEnd_Ext()
   LIN {X -1.758, Y -17.478, Z 107.100}
   LaserStart_Ext()
   LIN {X -3.810, Y -17.478, Z 107.100}
   LaserEnd_Ext()
   LIN {X -3.726, Y -18.478, Z 107.100}
   LaserStart_Ext()
   LIN {X -1.758, Y -18.478, Z 107.100}
   LaserEnd_Ext()
   LIN {X 9.911, Y -18.478, Z 107.100}
   LaserStart_Ext()
   LIN {X 11.959, Y -18.478, Z 107.100}
   LaserEnd_Ext()
   LIN {X 11.748, Y -19.478, Z 107.100}
   LaserStart_Ext()
   LIN {X 9.650, Y -19.478, Z 107.100}
   LaserEnd_Ext()
   LIN {X -1.426, Y -19.478, Z 107.100}
   LaserStart_Ext()
   LIN {X -3.456, Y -19.478, Z 107.100}
   LaserEnd_Ext()
   LIN {X -3.185, Y -20.478, Z 107.100}
   LaserStart_Ext()
   LIN {X -1.083, Y -20.478, Z 107.100}
   LaserEnd_Ext()
   LIN {X 9.262, Y -20.478, Z 107.100}
   LaserStart_Ext()
   LIN {X 11.449, Y -20.478, Z 107.100}
   LaserEnd_Ext()
   LIN {X 10.810, Y -21.478, Z 107.100}
   LaserStart_Ext()
   LIN {X 8.414, Y -21.478, Z 107.100}
   LaserEnd_Ext()
   LIN {X -0.212, Y -21.478, Z 107.100}
   LaserStart_Ext()
   LIN {X -2.750, Y -21.478, Z 107.100}
   LaserEnd_Ext()
   LIN {X -1.962, Y -22.478, Z 107.100}
   LaserStart_Ext()
   LIN {X 0.842, Y -22.478, Z 107.100}
   LaserEnd_Ext()
   LIN {X 7.262, Y -22.478, Z 107.100}
   LaserStart_Ext()
   LIN {X 10.170, Y -22.478, Z 107.100}
   LaserEnd_Ext()
   LIN {X 9.210, Y -23.478, Z 107.100}
   LaserStart_Ext()
   LIN {X -1.174, Y -23.478, Z 107.100}
   LaserEnd_Ext()
   LIN {X 0.538, Y -24.478, Z 107.100}
   LaserStart_Ext()
   LIN {X 7.752, Y -24.478, Z 107.100}
   LaserEnd_Ext()
   LIN {X 8.759, Y -15.276, Z 107.950}
   LaserStart_Ext()
   LIN {X 8.940, Y -16.152, Z 107.950} C_DIS
   LIN {X 9.211, Y -17.439, Z 107.950} C_DIS
   LIN {X 8.671, Y -19.520, Z 107.950} C_DIS
   LIN {X 8.617, Y -19.725, Z 107.950} C_DIS
   LIN {X 8.509, Y -19.852, Z 107.950} C_DIS
   LIN {X 7.233, Y -21.363, Z 107.950} C_DIS
   LIN {X 6.120, Y -21.883, Z 107.950} C_DIS
   LIN {X 5.268, Y -22.278, Z 107.950} C_DIS
   LIN {X 3.891, Y -22.301, Z 107.950} C_DIS
   LIN {X 3.211, Y -22.313, Z 107.950} C_DIS
   LIN {X 2.760, Y -22.122, Z 107.950} C_DIS
   LIN {X 1.311, Y -21.500, Z 107.950} C_DIS
   LIN {X -0.004, Y -20.086, Z 107.950} C_DIS
   LIN {X -0.108, Y -19.974, Z 107.950} C_DIS
   LIN {X -0.157, Y -19.829, Z 107.950} C_DIS
   LIN {X -0.768, Y -17.995, Z 107.950} C_DIS
   LIN {X -0.227, Y -15.201, Z 107.950} C_DIS
   LIN {X -0.193, Y -15.034, Z 107.950} C_DIS
   LIN {X -0.116, Y -14.945, Z 107.950} C_DIS
   LIN {X 1.197, Y -13.407, Z 107.950} C_DIS
   LIN {X 2.653, Y -12.736, Z 107.950} C_DIS
   LIN {X 3.146, Y -12.507, Z 107.950} C_DIS
   LIN {X 3.880, Y -12.493, Z 107.950} C_DIS
   LIN {X 5.189, Y -12.471, Z 107.950} C_DIS
   LIN {X 6.096, Y -12.866, Z 107.950} C_DIS
   LIN {X 7.140, Y -13.315, Z 107.950} C_DIS
   LIN {X 8.128, Y -14.509, Z 107.950} C_DIS
   LIN {X 8.759, Y -15.276, Z 107.950}
   LaserEnd_Ext()
   LIN {X -3.425, Y 45.265, Z 107.950}
   LaserStart_Ext()
   LIN {X -2.648, Y 44.003, Z 107.950} C_DIS
   LIN {X -1.938, Y 42.805, Z 107.950} C_DIS
   LIN {X -1.673, Y 42.354, Z 107.950} C_DIS
   LIN {X -1.311, Y 41.707, Z 107.950} C_DIS
   LIN {X -0.480, Y 40.227, Z 107.950} C_DIS
   LIN {X -0.057, Y 39.465, Z 107.950} C_DIS
   LIN {X 0.692, Y 38.020, Z 107.950} C_DIS
   LIN {X 1.594, Y 36.291, Z 107.950} C_DIS
   LIN {X 2.117, Y 35.196, Z 107.950} C_DIS
   LIN {X 3.786, Y 31.637, Z 107.950} C_DIS
   LIN {X 5.122, Y 28.352, Z 107.950} C_DIS
   LIN {X 6.606, Y 24.673, Z 107.950} C_DIS
   LIN {X 7.475, Y 22.021, Z 107.950} C_DIS
   LIN {X 8.938, Y 17.561, Z 107.950} C_DIS
   LIN {X 10.390, Y 11.654, Z 107.950} C_DIS
   LIN {X 11.273, Y 7.864, Z 107.950} C_DIS
   LIN {X 12.280, Y 1.227, Z 107.950} C_DIS
   LIN {X 12.589, Y -0.696, Z 107.950} C_DIS
   LIN {X 12.700, Y -1.864, Z 107.950} C_DIS
   LIN {X 13.105, Y -6.720, Z 107.950} C_DIS
   LIN {X 13.160, Y -7.668, Z 107.950} C_DIS
   LIN {X 13.259, Y -10.743, Z 107.950} C_DIS
   LIN {X 13.286, Y -11.472, Z 107.950} C_DIS
   LIN {X 13.288, Y -11.850, Z 107.950} C_DIS
   LIN {X 13.293, Y -14.431, Z 107.950} C_DIS
   LIN {X 13.239, Y -16.739, Z 107.950} C_DIS
   LIN {X 13.211, Y -17.693, Z 107.950} C_DIS
   LIN {X 12.929, Y -19.031, Z 107.950} C_DIS
   LIN {X 12.606, Y -20.592, Z 107.950} C_DIS
   LIN {X 12.042, Y -21.556, Z 107.950} C_DIS
   LIN {X 10.856, Y -23.410, Z 107.950} C_DIS
   LIN {X 9.280, Y -24.645, Z 107.950} C_DIS
   LIN {X 7.843, Y -25.619, Z 107.950} C_DIS
   LIN {X 5.939, Y -26.168, Z 107.950} C_DIS
   LIN {X 4.374, Y -26.244, Z 107.950} C_DIS
   LIN {X 1.654, Y -26.062, Z 107.950} C_DIS
   LIN {X -0.187, Y -25.151, Z 107.950} C_DIS
   LIN {X -1.608, Y -24.324, Z 107.950} C_DIS
   LIN {X -2.918, Y -22.662, Z 107.950} C_DIS
   LIN {X -3.825, Y -21.569, Z 107.950} C_DIS
   LIN {X -4.319, Y -19.780, Z 107.950} C_DIS
   LIN {X -4.803, Y -17.989, Z 107.950} C_DIS
   LIN {X -4.651, Y -16.731, Z 107.950} C_DIS
   LIN {X -4.431, Y -14.840, Z 107.950} C_DIS
   LIN {X -3.847, Y -12.742, Z 107.950} C_DIS
   LIN {X -3.604, Y -11.876, Z 107.950} C_DIS
   LIN {X -3.329, Y -10.666, Z 107.950} C_DIS
   LIN {X -2.811, Y -8.422, Z 107.950} C_DIS
   LIN {X -2.677, Y -7.767, Z 107.950} C_DIS
   LIN {X -1.856, Y -2.566, Z 107.950} C_DIS
   LIN {X -1.321, Y 6.932, Z 107.950} C_DIS
   LIN {X -1.730, Y 12.875, Z 107.950} C_DIS
   LIN {X -2.082, Y 16.693, Z 107.950} C_DIS
   LIN {X -3.146, Y 22.087, Z 107.950} C_DIS
   LIN {X -3.873, Y 25.265, Z 107.950} C_DIS
   LIN {X -5.249, Y 29.655, Z 107.950} C_DIS
   LIN {X -6.036, Y 31.949, Z 107.950} C_DIS
   LIN {X -7.486, Y 35.526, Z 107.950} C_DIS
   LIN {X -7.664, Y 35.926, Z 107.950} C_DIS
   LIN {X -7.766, Y 36.145, Z 107.950} C_DIS
   LIN {X -8.326, Y 37.338, Z 107.950} C_DIS
   LIN {X -8.983, Y 38.734, Z 107.950} C_DIS
   LIN {X -9.328, Y 39.410, Z 107.950} C_DIS
   LIN {X -9.710, Y 40.158, Z 107.950} C_DIS
   LIN {X -9.911, Y 40.542, Z 107.950} C_DIS
   LIN {X -10.294, Y 41.264, Z 107.950} C_DIS
   LIN {X -10.724, Y 42.561, Z 107.950} C_DIS
   LIN {X -10.760, Y 42.668, Z 107.950} C_DIS
   LIN {X -10.653, Y 44.236, Z 107.950} C_DIS
   LIN {X -9.900, Y 45.653, Z 107.950} C_DIS
   LIN {X -9.835, Y 45.774, Z 107.950} C_DIS
   LIN {X -9.517, Y 45.970, Z 107.950} C_DIS
   LIN {X -7.740, Y 47.052, Z 107.950} C_DIS
   LIN {X -6.594, Y 47.065, Z 107.950} C_DIS
   LIN {X -5.997, Y 47.072, Z 107.950} C_DIS
   LIN {X -5.632, Y 46.907, Z 107.950} C_DIS
   LIN {X -4.415, Y 46.352, Z 107.950} C_DIS
   LIN {X -3.426, Y 45.265, Z 107.950}
   LaserEnd_Ext()
   LIN {X -9.280, Y 41.486, Z 107.950}
   LaserStart_Ext()
   LIN {X -9.280, Y 44.688, Z 107.950}
   LaserEnd_Ext()
   LIN {X -8.280, Y 45.552, Z 107.950}
   LaserStart_Ext()
   LIN {X -8.280, Y 39.556, Z 107.950}
   LaserEnd_Ext()
   LIN {X -7.280, Y 37.462, Z 107.950}
   LaserStart_Ext()
   LIN {X -7.280, Y 46.057, Z 107.950}
   LaserEnd_Ext()
   LIN {X -6.280, Y 46.069, Z 107.950}
   LaserStart_Ext()
   LIN {X -6.280, Y 35.212, Z 107.950}
   LaserEnd_Ext()
   LIN {X -5.280, Y 32.747, Z 107.950}
   LaserStart_Ext()
   LIN {X -5.280, Y 45.648, Z 107.950}
   LaserEnd_Ext()
   LIN {X -4.280, Y 44.718, Z 107.950}
   LaserStart_Ext()
   LIN {X -4.280, Y 29.908, Z 107.950}
   LaserEnd_Ext()
   LIN {X -3.280, Y -19.786, Z 107.950}
   LaserStart_Ext()
   LIN {X -3.280, Y -14.433, Z 107.950}
   LaserEnd_Ext()
   LIN {X -3.280, Y 26.716, Z 107.950}
   LaserStart_Ext()
   LIN {X -3.280, Y 43.107, Z 107.950}
   LaserEnd_Ext()
   LIN {X -2.280, Y 41.390, Z 107.950}
   LaserStart_Ext()
   LIN {X -2.280, Y 22.784, Z 107.950}
   LaserEnd_Ext()
   LIN {X -2.280, Y -10.567, Z 107.950}
   LaserStart_Ext()
   LIN {X -2.280, Y -21.865, Z 107.950}
   LaserEnd_Ext()
   LIN {X -1.280, Y -23.125, Z 107.950}
   LaserStart_Ext()
   LIN {X -1.280, Y -19.623, Z 107.950}
   LaserEnd_Ext()
   LIN {X -1.280, Y -15.378, Z 107.950}
   LaserStart_Ext()
   LIN {X -1.280, Y -5.329, Z 107.950}
   LaserEnd_Ext()
   LIN {X -1.280, Y 17.795, Z 107.950}
   LaserStart_Ext()
   LIN {X -1.280, Y 39.607, Z 107.950}
   LaserEnd_Ext()
   LIN {X -0.280, Y 37.723, Z 107.950}
   LaserStart_Ext()
   LIN {X -0.280, Y -13.597, Z 107.950}
   LaserEnd_Ext()
   LIN {X -0.280, Y -21.258, Z 107.950}
   LaserStart_Ext()
   LIN {X -0.280, Y -23.940, Z 107.950}
   LaserEnd_Ext()
   LIN {X 0.720, Y -24.484, Z 107.950}
   LaserStart_Ext()
   LIN {X 0.720, Y -22.306, Z 107.950}
   LaserEnd_Ext()
   LIN {X 0.720, Y -12.530, Z 107.950}
   LaserStart_Ext()
   LIN {X 0.720, Y 35.799, Z 107.950}
   LaserEnd_Ext()
   LIN {X 1.720, Y 33.688, Z 107.950}
   LaserStart_Ext()
   LIN {X 1.720, Y -12.065, Z 107.950}
   LaserEnd_Ext()
   LIN {X 1.720, Y -22.764, Z 107.950}
   LaserStart_Ext()
   LIN {X 1.720, Y -24.979, Z 107.950}
   LaserEnd_Ext()
   LIN {X 2.720, Y -25.131, Z 107.950}
   LaserStart_Ext()
   LIN {X 2.720, Y -23.191, Z 107.950}
   LaserEnd_Ext()
   LIN {X 2.720, Y -11.602, Z 107.950}
   LaserStart_Ext()
   LIN {X 2.720, Y 31.555, Z 107.950}
   LaserEnd_Ext()
   LIN {X 3.720, Y 29.145, Z 107.950}
   LaserStart_Ext()
   LIN {X 3.720, Y -11.496, Z 107.950}
   LaserEnd_Ext()
   LIN {X 3.720, Y -23.305, Z 107.950}
   LaserStart_Ext()
   LIN {X 3.720, Y -25.198, Z 107.950}
   LaserEnd_Ext()
   LIN {X 4.720, Y -25.226, Z 107.950}
   LaserStart_Ext()
   LIN {X 4.720, Y -23.288, Z 107.950}
   LaserEnd_Ext()
   LIN {X 4.720, Y -11.479, Z 107.950}
   LaserStart_Ext()
   LIN {X 4.720, Y 26.675, Z 107.950}
   LaserEnd_Ext()
   LIN {X 5.720, Y 24.163, Z 107.950}
   LaserStart_Ext()
   LIN {X 5.720, Y -11.611, Z 107.950}
   LaserEnd_Ext()
   LIN {X 5.720, Y -23.171, Z 107.950}
   LaserStart_Ext()
   LIN {X 5.720, Y -25.178, Z 107.950}
   LaserEnd_Ext()
   LIN {X 6.720, Y -24.902, Z 107.950}
   LaserStart_Ext()
   LIN {X 6.720, Y -22.706, Z 107.950}
   LaserEnd_Ext()
   LIN {X 6.720, Y -12.046, Z 107.950}
   LaserStart_Ext()
   LIN {X 6.720, Y 21.113, Z 107.950}
   LaserEnd_Ext()
   LIN {X 7.720, Y 18.065, Z 107.950}
   LaserStart_Ext()
   LIN {X 7.720, Y -12.502, Z 107.950}
   LaserEnd_Ext()
   LIN {X 7.720, Y -22.235, Z 107.950}
   LaserStart_Ext()
   LIN {X 7.720, Y -24.494, Z 107.950}
   LaserEnd_Ext()
   LIN {X 8.720, Y -23.813, Z 107.950}
   LaserStart_Ext()
   LIN {X 8.720, Y -21.152, Z 107.950}
   LaserEnd_Ext()
   LIN {X 8.720, Y -13.656, Z 107.950}
   LaserStart_Ext()
   LIN {X 8.720, Y 14.258, Z 107.950}
   LaserEnd_Ext()
   LIN {X 9.720, Y 10.122, Z 107.950}
   LaserStart_Ext()
   LIN {X 9.720, Y -15.004, Z 107.950}
   LaserEnd_Ext()
   LIN {X 9.720, Y -19.457, Z 107.950}
   LaserStart_Ext()
   LIN {X 9.720, Y -23.030, Z 107.950}
   LaserEnd_Ext()
   LIN {X 10.720, Y -21.767, Z 107.950}
   LaserStart_Ext()
   LIN {X 10.720, Y 4.842, Z 107.950}
   LaserEnd_Ext()
   LIN {X 11.720, Y -2.141, Z 107.950}
   LaserStart_Ext()
   LIN {X 11.720, Y -19.937, Z 107.950}
   LaserEnd_Ext()
   LIN {X 1.270, Y -13.352, Z 108.800}
   LaserStart_Ext()
   LIN {X 1.544, Y -13.226, Z 108.800} C_DIS
   LIN {X 3.214, Y -12.449, Z 108.800} C_DIS
   LIN {X 4.934, Y -12.416, Z 108.800} C_DIS
   LIN {X 5.258, Y -12.409, Z 108.800} C_DIS
   LIN {X 5.661, Y -12.581, Z 108.800} C_DIS
   LIN {X 7.210, Y -13.249, Z 108.800} C_DIS
   LIN {X 8.320, Y -14.589, Z 108.800} C_DIS
   LIN {X 8.834, Y -15.206, Z 108.800} C_DIS
   LIN {X 8.964, Y -15.813, Z 108.800} C_DIS
   LIN {X 9.291, Y -17.368, Z 108.800} C_DIS
   LIN {X 8.961, Y -18.639, Z 108.800} C_DIS
   LIN {X 8.699, Y -19.661, Z 108.800} C_DIS
   LIN {X 7.951, Y -20.551, Z 108.800} C_DIS
   LIN {X 7.322, Y -21.296, Z 108.800} C_DIS
   LIN {X 5.858, Y -21.979, Z 108.800} C_DIS
   LIN {X 5.350, Y -22.218, Z 108.800} C_DIS
   LIN {X 5.011, Y -22.225, Z 108.800} C_DIS
   LIN {X 3.302, Y -22.256, Z 108.800} C_DIS
   LIN {X 1.614, Y -21.538, Z 108.800} C_DIS
   LIN {X 1.399, Y -21.446, Z 108.800} C_DIS
   LIN {X 1.205, Y -21.237, Z 108.800} C_DIS
   LIN {X -0.023, Y -19.924, Z 108.800} C_DIS
   LIN {X -0.597, Y -18.217, Z 108.800} C_DIS
   LIN {X -0.688, Y -17.946, Z 108.800} C_DIS
   LIN {X -0.596, Y -17.473, Z 108.800} C_DIS
   LIN {X -0.118, Y -14.983, Z 108.800} C_DIS
   LIN {X 0.989, Y -13.682, Z 108.800} C_DIS
   LIN {X 1.270, Y -13.352, Z 108.800}
   LaserEnd_Ext()
   LIN {X -6.069, Y 47.107, Z 108.800}
   LaserStart_Ext()
   LIN {X -4.651, Y 46.466, Z 108.800} C_DIS
   LIN {X -4.485, Y 46.391, Z 108.800} C_DIS
   LIN {X -4.402, Y 46.300, Z 108.800} C_DIS
   LIN {X -3.495, Y 45.306, Z 108.800} C_DIS
   LIN {X -2.809, Y 44.203, Z 108.800} C_DIS
   LIN {X -2.712, Y 44.046, Z 108.800} C_DIS
   LIN {X -2.542, Y 43.759, Z 108.800} C_DIS
   LIN {X -1.771, Y 42.462, Z 108.800} C_DIS
   LIN {X -1.595, Y 42.160, Z 108.800} C_DIS
   LIN {X -0.782, Y 40.712, Z 108.800} C_DIS
   LIN {X 0.086, Y 39.150, Z 108.800} C_DIS
   LIN {X 1.621, Y 36.190, Z 108.800} C_DIS
   LIN {X 1.752, Y 35.939, Z 108.800} C_DIS
   LIN {X 1.828, Y 35.780, Z 108.800} C_DIS
   LIN {X 3.908, Y 31.345, Z 108.800} C_DIS
   LIN {X 4.989, Y 28.686, Z 108.800} C_DIS
   LIN {X 6.657, Y 24.549, Z 108.800} C_DIS
   LIN {X 7.372, Y 22.366, Z 108.800} C_DIS
   LIN {X 9.028, Y 17.322, Z 108.800} C_DIS
   LIN {X 10.245, Y 12.366, Z 108.800} C_DIS
   LIN {X 11.392, Y 7.448, Z 108.800} C_DIS
   LIN {X 12.669, Y -0.974, Z 108.800} C_DIS
   LIN {X 12.771, Y -2.161, Z 108.800} C_DIS
   LIN {X 13.207, Y -7.386, Z 108.800} C_DIS
   LIN {X 13.218, Y -7.587, Z 108.800} C_DIS
   LIN {X 13.239, Y -8.242, Z 108.800} C_DIS
   LIN {X 13.354, Y -11.390, Z 108.800} C_DIS
   LIN {X 13.364, Y -13.026, Z 108.800} C_DIS
   LIN {X 13.367, Y -14.350, Z 108.800} C_DIS
   LIN {X 13.303, Y -17.060, Z 108.800} C_DIS
   LIN {X 13.292, Y -17.612, Z 108.800} C_DIS
   LIN {X 13.238, Y -17.880, Z 108.800} C_DIS
   LIN {X 12.694, Y -20.512, Z 108.800} C_DIS
   LIN {X 11.514, Y -22.530, Z 108.800} C_DIS
   LIN {X 11.110, Y -23.163, Z 108.800} C_DIS
   LIN {X 8.871, Y -24.917, Z 108.800} C_DIS
   LIN {X 7.924, Y -25.559, Z 108.800} C_DIS
   LIN {X 5.769, Y -26.181, Z 108.800} C_DIS
   LIN {X 5.430, Y -26.272, Z 108.800} C_DIS
   LIN {X 5.179, Y -26.255, Z 108.800} C_DIS
   LIN {X 1.838, Y -26.030, Z 108.800} C_DIS
   LIN {X -0.871, Y -24.690, Z 108.800} C_DIS
   LIN {X -1.381, Y -24.394, Z 108.800} C_DIS
   LIN {X -1.851, Y -23.797, Z 108.800} C_DIS
   LIN {X -3.735, Y -21.527, Z 108.800} C_DIS
   LIN {X -4.700, Y -18.027, Z 108.800} C_DIS
   LIN {X -4.710, Y -17.836, Z 108.800} C_DIS
   LIN {X -4.357, Y -14.800, Z 108.800} C_DIS
   LIN {X -3.723, Y -12.523, Z 108.800} C_DIS
   LIN {X -3.538, Y -11.835, Z 108.800} C_DIS
   LIN {X -2.857, Y -8.887, Z 108.800} C_DIS
   LIN {X -2.601, Y -7.629, Z 108.800} C_DIS
   LIN {X -1.906, Y -3.230, Z 108.800} C_DIS
   LIN {X -1.815, Y -2.605, Z 108.800} C_DIS
   LIN {X -1.734, Y -1.159, Z 108.800} C_DIS
   LIN {X -1.294, Y 6.682, Z 108.800} C_DIS
   LIN {X -1.754, Y 13.369, Z 108.800} C_DIS
   LIN {X -2.037, Y 16.443, Z 108.800} C_DIS
   LIN {X -3.223, Y 22.455, Z 108.800} C_DIS
   LIN {X -3.790, Y 24.932, Z 108.800} C_DIS
   LIN {X -5.434, Y 30.179, Z 108.800} C_DIS
   LIN {X -5.907, Y 31.559, Z 108.800} C_DIS
   LIN {X -7.064, Y 34.411, Z 108.800} C_DIS
   LIN {X -7.457, Y 35.392, Z 108.800} C_DIS
   LIN {X -7.618, Y 35.764, Z 108.800} C_DIS
   LIN {X -8.209, Y 37.007, Z 108.800} C_DIS
   LIN {X -9.034, Y 38.762, Z 108.800} C_DIS
   LIN {X -9.433, Y 39.542, Z 108.800} C_DIS
   LIN {X -9.765, Y 40.184, Z 108.800} C_DIS
   LIN {X -10.225, Y 41.051, Z 108.800} C_DIS
   LIN {X -10.351, Y 41.289, Z 108.800} C_DIS
   LIN {X -10.420, Y 41.495, Z 108.800} C_DIS
   LIN {X -10.819, Y 42.681, Z 108.800} C_DIS
   LIN {X -10.709, Y 44.256, Z 108.800} C_DIS
   LIN {X -9.927, Y 45.773, Z 108.800} C_DIS
   LIN {X -8.502, Y 46.648, Z 108.800} C_DIS
   LIN {X -7.811, Y 47.083, Z 108.800} C_DIS
   LIN {X -7.145, Y 47.093, Z 108.800} C_DIS
   LIN {X -6.069, Y 47.107, Z 108.800}
   LaserEnd_Ext()
   LIN {X 7.910, Y -24.360, Z 108.800}
   LaserStart_Ext()
   LIN {X 0.717, Y -24.360, Z 108.800}
   LaserEnd_Ext()
   LIN {X -0.922, Y -23.360, Z 108.800}
   LaserStart_Ext()
   LIN {X 9.237, Y -23.360, Z 108.800}
   LaserEnd_Ext()
   LIN {X 10.436, Y -22.360, Z 108.800}
   LaserStart_Ext()
   LIN {X 7.407, Y -22.360, Z 108.800}
   LaserEnd_Ext()
   LIN {X 0.994, Y -22.360, Z 108.800}
   LaserStart_Ext()
   LIN {X -1.744, Y -22.360, Z 108.800}
   LaserEnd_Ext()
   LIN {X -2.574, Y -21.360, Z 108.800}
   LaserStart_Ext()
   LIN {X -0.049, Y -21.360, Z 108.800}
   LaserEnd_Ext()
   LIN {X 8.577, Y -21.360, Z 108.800}
   LaserStart_Ext()
   LIN {X 11.040, Y -21.360, Z 108.800}
   LaserEnd_Ext()
   LIN {X 11.625, Y -20.360, Z 108.800}
   LaserStart_Ext()
   LIN {X 9.418, Y -20.360, Z 108.800}
   LaserEnd_Ext()
   LIN {X -0.922, Y -20.360, Z 108.800}
   LaserStart_Ext()
   LIN {X -3.020, Y -20.360, Z 108.800}
   LaserEnd_Ext()
   LIN {X -3.295, Y -19.360, Z 108.800}
   LaserStart_Ext()
   LIN {X -1.268, Y -19.360, Z 108.800}
   LaserEnd_Ext()
   LIN {X 9.808, Y -19.360, Z 108.800}
   LaserStart_Ext()
   LIN {X 11.911, Y -19.360, Z 108.800}
   LaserEnd_Ext()
   LIN {X 12.118, Y -18.360, Z 108.800}
   LaserStart_Ext()
   LIN {X 10.066, Y -18.360, Z 108.800}
   LaserEnd_Ext()
   LIN {X -1.604, Y -18.360, Z 108.800}
   LaserStart_Ext()
   LIN {X -3.571, Y -18.360, Z 108.800}
   LaserEnd_Ext()
   LIN {X -3.647, Y -17.360, Z 108.800}
   LaserStart_Ext()
   LIN {X -1.593, Y -17.360, Z 108.800}
   LaserEnd_Ext()
   LIN {X 10.290, Y -17.360, Z 108.800}
   LaserStart_Ext()
   LIN {X 12.297, Y -17.360, Z 108.800}
   LaserEnd_Ext()
   LIN {X 12.320, Y -16.360, Z 108.800}
   LaserStart_Ext()
   LIN {X 10.101, Y -16.360, Z 108.800}
   LaserEnd_Ext()
   LIN {X -1.401, Y -16.360, Z 108.800}
   LaserStart_Ext()
   LIN {X -3.531, Y -16.360, Z 108.800}
   LaserEnd_Ext()
   LIN {X -3.415, Y -15.360, Z 108.800}
   LaserStart_Ext()
   LIN {X -1.209, Y -15.360, Z 108.800}
   LaserEnd_Ext()
   LIN {X 9.890, Y -15.360, Z 108.800}
   LaserStart_Ext()
   LIN {X 12.343, Y -15.360, Z 108.800}
   LaserEnd_Ext()
   LIN {X 12.366, Y -14.360, Z 108.800}
   LaserStart_Ext()
   LIN {X 9.431, Y -14.360, Z 108.800}
   LaserEnd_Ext()
   LIN {X -0.899, Y -14.360, Z 108.800}
   LaserStart_Ext()
   LIN {X -3.196, Y -14.360, Z 108.800}
   LaserEnd_Ext()
   LIN {X -2.918, Y -13.360, Z 108.800}
   LaserStart_Ext()
   LIN {X -0.050, Y -13.360, Z 108.800}
   LaserEnd_Ext()
   LIN {X 8.601, Y -13.360, Z 108.800}
   LaserStart_Ext()
   LIN {X 12.365, Y -13.360, Z 108.800}
   LaserEnd_Ext()
   LIN {X 12.360, Y -12.360, Z 108.800}
   LaserStart_Ext()
   LIN {X 7.667, Y -12.360, Z 108.800}
   LaserEnd_Ext()
   LIN {X 1.033, Y -12.360, Z 108.800}
   LaserStart_Ext()
   LIN {X -2.644, Y -12.360, Z 108.800}
   LaserEnd_Ext()
   LIN {X -2.402, Y -11.360, Z 108.800}
   LaserStart_Ext()
   LIN {X 12.352, Y -11.360, Z 108.800}
   LaserEnd_Ext()
   LIN {X 12.316, Y -10.360, Z 108.800}
   LaserStart_Ext()
   LIN {X -2.171, Y -10.360, Z 108.800}
   LaserEnd_Ext()
   LIN {X -1.940, Y -9.360, Z 108.800}
   LaserStart_Ext()
   LIN {X 12.279, Y -9.360, Z 108.800}
   LaserEnd_Ext()
   LIN {X 12.243, Y -8.360, Z 108.800}
   LaserStart_Ext()
   LIN {X -1.729, Y -8.360, Z 108.800}
   LaserEnd_Ext()
   LIN {X -1.546, Y -7.360, Z 108.800}
   LaserStart_Ext()
   LIN {X 12.201, Y -7.360, Z 108.800}
   LaserEnd_Ext()
   LIN {X 12.118, Y -6.360, Z 108.800}
   LaserStart_Ext()
   LIN {X -1.388, Y -6.360, Z 108.800}
   LaserEnd_Ext()
   LIN {X -1.230, Y -5.360, Z 108.800}
   LaserStart_Ext()
   LIN {X 12.034, Y -5.360, Z 108.800}
   LaserEnd_Ext()
   LIN {X 11.951, Y -4.360, Z 108.800}
   LaserStart_Ext()
   LIN {X -1.072, Y -4.360, Z 108.800}
   LaserEnd_Ext()
   LIN {X -0.914, Y -3.360, Z 108.800}
   LaserStart_Ext()
   LIN {X 11.868, Y -3.360, Z 108.800}
   LaserEnd_Ext()
   LIN {X 11.784, Y -2.360, Z 108.800}
   LaserStart_Ext()
   LIN {X -0.799, Y -2.360, Z 108.800}
   LaserEnd_Ext()
   LIN {X -0.743, Y -1.360, Z 108.800}
   LaserStart_Ext()
   LIN {X 11.702, Y -1.360, Z 108.800}
   LaserEnd_Ext()
   LIN {X 11.565, Y -0.360, Z 108.800}
   LaserStart_Ext()
   LIN {X -0.687, Y -0.360, Z 108.800}
   LaserEnd_Ext()
   LIN {X -0.631, Y 0.640, Z 108.800}
   LaserStart_Ext()
   LIN {X 11.413, Y 0.640, Z 108.800}
   LaserEnd_Ext()
   LIN {X 11.261, Y 1.640, Z 108.800}
   LaserStart_Ext()
   LIN {X -0.575, Y 1.640, Z 108.800}
   LaserEnd_Ext()
   LIN {X -0.519, Y 2.640, Z 108.800}
   LaserStart_Ext()
   LIN {X 11.110, Y 2.640, Z 108.800}
   LaserEnd_Ext()
   LIN {X 10.958, Y 3.640, Z 108.800}
   LaserStart_Ext()
   LIN {X -0.463, Y 3.640, Z 108.800}
   LaserEnd_Ext()
   LIN {X -0.407, Y 4.640, Z 108.800}
   LaserStart_Ext()
   LIN {X 10.807, Y 4.640, Z 108.800}
   LaserEnd_Ext()
   LIN {X 10.655, Y 5.640, Z 108.800}
   LaserStart_Ext()
   LIN {X -0.350, Y 5.640, Z 108.800}
   LaserEnd_Ext()
   LIN {X -0.295, Y 6.640, Z 108.800}
   LaserStart_Ext()
   LIN {X 10.503, Y 6.640, Z 108.800}
   LaserEnd_Ext()
   LIN {X 10.321, Y 7.640, Z 108.800}
   LaserStart_Ext()
   LIN {X -0.357, Y 7.640, Z 108.800}
   LaserEnd_Ext()
   LIN {X -0.426, Y 8.640, Z 108.800}
   LaserStart_Ext()
   LIN {X 10.088, Y 8.640, Z 108.800}
   LaserEnd_Ext()
   LIN {X 9.854, Y 9.640, Z 108.800}
   LaserStart_Ext()
   LIN {X -0.495, Y 9.640, Z 108.800}
   LaserEnd_Ext()
   LIN {X -0.563, Y 10.640, Z 108.800}
   LaserStart_Ext()
   LIN {X 9.621, Y 10.640, Z 108.800}
   LaserEnd_Ext()
   LIN {X 9.388, Y 11.640, Z 108.800}
   LaserStart_Ext()
   LIN {X -0.632, Y 11.640, Z 108.800}
   LaserEnd_Ext()
   LIN {X -0.701, Y 12.640, Z 108.800}
   LaserStart_Ext()
   LIN {X 9.148, Y 12.640, Z 108.800}
   LaserEnd_Ext()
   LIN {X 8.903, Y 13.640, Z 108.800}
   LaserStart_Ext()
   LIN {X -0.774, Y 13.640, Z 108.800}
   LaserEnd_Ext()
   LIN {X -0.866, Y 14.640, Z 108.800}
   LaserStart_Ext()
   LIN {X 8.657, Y 14.640, Z 108.800}
   LaserEnd_Ext()
   LIN {X 8.411, Y 15.640, Z 108.800}
   LaserStart_Ext()
   LIN {X -0.959, Y 15.640, Z 108.800}
   LaserEnd_Ext()
   LIN {X -1.056, Y 16.640, Z 108.800}
   LaserStart_Ext()
   LIN {X 8.165, Y 16.640, Z 108.800}
   LaserEnd_Ext()
   LIN {X 7.871, Y 17.640, Z 108.800}
   LaserStart_Ext()
   LIN {X -1.254, Y 17.640, Z 108.800}
   LaserEnd_Ext()
   LIN {X -1.451, Y 18.640, Z 108.800}
   LaserStart_Ext()
   LIN {X 7.543, Y 18.640, Z 108.800}
   LaserEnd_Ext()
   LIN {X 7.214, Y 19.640, Z 108.800}
   LaserStart_Ext()
   LIN {X -1.648, Y 19.640, Z 108.800}
   LaserEnd_Ext()
   LIN {X -1.846, Y 20.640, Z 108.800}
   LaserStart_Ext()
   LIN {X 6.886, Y 20.640, Z 108.800}
   LaserEnd_Ext()
   LIN {X 6.558, Y 21.640, Z 108.800}
   LaserStart_Ext()
   LIN {X -2.043, Y 21.640, Z 108.800}
   LaserEnd_Ext()
   LIN {X -2.241, Y 22.640, Z 108.800}
   LaserStart_Ext()
   LIN {X 6.230, Y 22.640, Z 108.800}
   LaserEnd_Ext()
   LIN {X 5.903, Y 23.640, Z 108.800}
   LaserStart_Ext()
   LIN {X -2.469, Y 23.640, Z 108.800}
   LaserEnd_Ext()
